			(* Case 60 - AspirazioneDX *)
			60: 
				IF AspirazioneSX^.Status.CommandDone AND AspirazioneDX^.Status.CommandDone THEN
					AspirazioneDX^.Command^.Aspirazione_ON 	:= FALSE;
					AspirazioneDX^.Command^.Aspirazione_OFF	:= FALSE;
					AspirazioneSX^.Command^.Aspirazione_ON 	:= FALSE;
					AspirazioneSX^.Command^.Aspirazione_OFF	:= FALSE;
					TFCommandCase(ADR(CmdExe),100,CommandCase_JMP);
				ELSIF AspirazioneSX^.Status.ErrorID <> ErrNULL THEN
					TFClearAllCmdModulePinzaCompleta(AspirazioneDX,AspirazioneSX,CilindroApertura,CilindroSbloccoRotazione,AspirazioneFaldaDX,AspirazioneFaldaSX);
					TFError(ErrCYLINDER,AspirazioneSX^.Status.ErrorID,ADR(CmdExe),ADR(State),ADR(Error),ADR(ErrorLog));
				ELSIF AspirazioneDX^.Status.ErrorID <> ErrNULL THEN
					TFClearAllCmdModulePinzaCompleta(AspirazioneDX,AspirazioneSX,CilindroApertura,CilindroSbloccoRotazione,AspirazioneFaldaDX,AspirazioneFaldaSX);
					TFError(ErrCYLINDER,AspirazioneDX^.Status.ErrorID,ADR(CmdExe),ADR(State),ADR(Error),ADR(ErrorLog));
				END_IF

			(* Case 70 - CilindroTasteggio *)
			70: 
				//IF CilindroTasteggio^.Status.CommandDone THEN
				//	CilindroTasteggio^.Command.Activation 		:= FALSE;
				//	CilindroTasteggio^.Command.Deactivation 	:= FALSE;
					TFCommandCase(ADR(CmdExe),100,CommandCase_JMP);
				//END_IF								
				
			(* Case 100 - End *)
			100:(* Clear All Output Here *)
				TFStateUpdate(ADR(State),StateMAN_END);
				TFCommandExeClear(ADR(CmdExe));

			ELSE
				TFError(ErrNOCMDCASE,ErrNULL,ADR(CmdExe),ADR(State),ADR(Error),ADR(ErrorLog));
		END_CASE;

		IF TFTimerDone(ADR(Timeout)) THEN
			TFClearAllCmdModulePinzaCompleta(AspirazioneDX,AspirazioneSX,CilindroApertura,CilindroSbloccoRotazione,AspirazioneFaldaDX,AspirazioneFaldaSX);
			TFError(ErrCMDTIMEOUT,ErrNULL,ADR(CmdExe),ADR(State),ADR(Error),ADR(ErrorLog));
		END_IF
	

	(* ******************************************************************************************************** *)
	(* PRELOAD - Presa del pezzo *)
	(* ******************************************************************************************************** *)
	CmdPRELOAD:
		CASE CmdExe.CmdCase OF
			
			(* Case 0 - Init Command*)
			0: 	TFStateUpdate(ADR(State),StatePRELOAD_RUN);
				TFTimerSet(ADR(Timeout),30000+200,TRUE);
				TFTimerSet(ADR(Timer),30000,TRUE);
				PrelievoSuCavallina := FALSE;
				StatoPinza.ElementoPrelevato := FALSE;
				IF TFCommandParRead(CmdExe.Cmd.Parameter,ADR(ParametersArray),2) THEN
					PrelievoSuCavallina	:= STRING_TO_BOOL(ParametersArray.Parameters[0]);
					AspiraSoloFalde		:= STRING_TO_BOOL(ParametersArray.Parameters[1]);
					TFCommandCase(ADR(CmdExe),10,CommandCase_JMP);
				ELSE
					TFError(ErrCMDPARNUM,ErrNULL,ADR(CmdExe),ADR(State),ADR(Error),ADR(ErrorLog));
					RETURN;
				END_IF;
				
			(* Case 10 - CilindroApertura *)
			10: 
				IF (ElementoInPrelievo.Typology = QUADROTTA OR ElementoInPrelievo.XDim >= 2700) AND AbilitaAperturaAutomaticaPinza THEN //sE HO LE CONDIZIONI APRO LA PINZA
					CilindroApertura^.Command.Activation 	:= TRUE;
					CilindroApertura^.Command.Deactivation 	:= FALSE;
	
					IF CilindroApertura^.Status.Active THEN
						CilindroApertura^.Command.Activation 	:= FALSE;
						CilindroApertura^.Command.Deactivation 	:= FALSE;
						TFCommandCase(ADR(CmdExe),20,CommandCase_JMP);
					ELSIF CilindroApertura^.Status.ErrorID <> ErrNULL THEN
						TFClearAllCmdModulePinzaCompleta(AspirazioneDX,AspirazioneSX,CilindroApertura,CilindroSbloccoRotazione,AspirazioneFaldaDX,AspirazioneFaldaSX);
						TFError(ErrCYLINDER,CilindroApertura^.Status.ErrorID,ADR(CmdExe),ADR(State),ADR(Error),ADR(ErrorLog));
					END_IF
				ELSE

					CilindroApertura^.Command.Activation 	:= FALSE;
					CilindroApertura^.Command.Deactivation 	:= TRUE;
	
					IF CilindroApertura^.Status.Inactive THEN
						CilindroApertura^.Command.Activation 	:= FALSE;
						CilindroApertura^.Command.Deactivation 	:= FALSE;
						TFCommandCase(ADR(CmdExe),20,CommandCase_JMP);
					ELSIF CilindroApertura^.Status.ErrorID <> ErrNULL THEN
						TFClearAllCmdModulePinzaCompleta(AspirazioneDX,AspirazioneSX,CilindroApertura,CilindroSbloccoRotazione,AspirazioneFaldaDX,AspirazioneFaldaSX);
						TFError(ErrCYLINDER,CilindroApertura^.Status.ErrorID,ADR(CmdExe),ADR(State),ADR(Error),ADR(ErrorLog));
					END_IF
					
				END_IF

			(* Case 20 - CilindroSbloccoRotazione *)
			20: 
				IF PrelievoSuCavallina THEN
					CilindroSbloccoRotazione^.Command.Activation 	:= AbilitazioneSbloccoRotazione;
					CilindroSbloccoRotazione^.Command.Deactivation 	:= FALSE;
	
					//CilindroTasteggio^.Command.Activation 		:= AbilitazioneCilindriTastatori;
					//CilindroTasteggio^.Command.Deactivation 	:= FALSE;
					
					IF (CilindroSbloccoRotazione^.Status.Active OR NOT AbilitazioneSbloccoRotazione) THEN
						CilindroSbloccoRotazione^.Command.Activation 	:= FALSE;
						CilindroSbloccoRotazione^.Command.Deactivation 	:= FALSE;
						//CilindroTasteggio^.Command.Activation 		:= FALSE;
						//CilindroTasteggio^.Command.Deactivation 	:= FALSE;
						TFCommandCase(ADR(CmdExe),30,CommandCase_JMP);
					ELSIF CilindroSbloccoRotazione^.Status.ErrorID <> ErrNULL AND AbilitazioneSbloccoRotazione THEN
						TFClearAllCmdModulePinzaCompleta(AspirazioneDX,AspirazioneSX,CilindroApertura,CilindroSbloccoRotazione,AspirazioneFaldaDX,AspirazioneFaldaSX);
						TFError(ErrCYLINDER,CilindroSbloccoRotazione^.Status.ErrorID,ADR(CmdExe),ADR(State),ADR(Error),ADR(ErrorLog));
					//ELSIF CilindroTasteggio^.Status.ErrorID <> ErrNULL THEN
					//	TFClearAllCmdModulePinzaCompleta(AspirazioneDX,AspirazioneSX,CilindroApertura,CilindroSbloccoRotazione,AspirazioneFaldaDX,AspirazioneFaldaSX);
					//	TFError(ErrCYLINDER,CilindroTasteggio^.Status.ErrorID,ADR(CmdExe),ADR(State),ADR(Error),ADR(ErrorLog));
					END_IF

				ELSE
					TFCommandCase(ADR(CmdExe),30,CommandCase_JMP);
				END_IF

			(* Case 30 - AspirazioneFaldaDX *)
			30: 

				IF NOT PrelievoSuCavallina AND AspiraSoloFalde THEN
					AspirazioneFaldaDX^.Command.Activation 	:= TRUE;
					AspirazioneFaldaDX^.Command.Deactivation 	:= FALSE;
					AspirazioneFaldaSX^.Command.Activation 	:= TRUE;
					AspirazioneFaldaSX^.Command.Deactivation 	:= FALSE;
					
					IF AspirazioneFaldaDX^.Status.Active AND AspirazioneFaldaSX^.Status.Active THEN
						AspirazioneFaldaDX^.Command.Activation 	:= FALSE;
						AspirazioneFaldaDX^.Command.Deactivation 	:= FALSE;
						AspirazioneFaldaSX^.Command.Activation 	:= FALSE;
						AspirazioneFaldaSX^.Command.Deactivation 	:= FALSE;
						TFCommandCase(ADR(CmdExe),40,CommandCase_JMP);
					ELSIF AspirazioneFaldaDX^.Status.ErrorID <> ErrNULL THEN
						TFClearAllCmdModulePinzaCompleta(AspirazioneDX,AspirazioneSX,CilindroApertura,CilindroSbloccoRotazione,AspirazioneFaldaDX,AspirazioneFaldaSX);
						TFError(ErrCYLINDER,AspirazioneFaldaDX^.Status.ErrorID,ADR(CmdExe),ADR(State),ADR(Error),ADR(ErrorLog));
					ELSIF AspirazioneFaldaSX^.Status.ErrorID <> ErrNULL THEN
						TFClearAllCmdModulePinzaCompleta(AspirazioneDX,AspirazioneSX,CilindroApertura,CilindroSbloccoRotazione,AspirazioneFaldaDX,AspirazioneFaldaSX);
						TFError(ErrCYLINDER,AspirazioneFaldaSX^.Status.ErrorID,ADR(CmdExe),ADR(State),ADR(Error),ADR(ErrorLog));
					END_IF
				ELSE
					TFCommandCase(ADR(CmdExe),40,CommandCase_JMP);
				END_IF


			(* Case 40 - AspirazioneDX + AspirazioneSX *)
			40: 
				AspirazioneDX^.Command^.Aspirazione_ON 	:= TRUE;
				AspirazioneDX^.Command^.Aspirazione_OFF := FALSE;
			
				AspirazioneSX^.Command^.Aspirazione_ON 	:= TRUE;
				AspirazioneSX^.Command^.Aspirazione_OFF := FALSE;
	
				IF AspirazioneDX^.Status.CommandDone AND AspirazioneSX^.Status.CommandDone THEN
					AspirazioneDX^.Command^.Aspirazione_ON 	:= FALSE;
					AspirazioneDX^.Command^.Aspirazione_OFF	:= FALSE;
					AspirazioneSX^.Command^.Aspirazione_ON 	:= FALSE;
					AspirazioneSX^.Command^.Aspirazione_OFF	:= FALSE;
					TFCommandCase(ADR(CmdExe),100,CommandCase_JMP);
				ELSIF AspirazioneSX^.Status.ErrorID <> ErrNULL THEN
					TFClearAllCmdModulePinzaCompleta(AspirazioneDX,AspirazioneSX,CilindroApertura,CilindroSbloccoRotazione,AspirazioneFaldaDX,AspirazioneFaldaSX);
					TFError(ErrCYLINDER,AspirazioneSX^.Status.ErrorID,ADR(CmdExe),ADR(State),ADR(Error),ADR(ErrorLog));
				ELSIF AspirazioneDX^.Status.ErrorID <> ErrNULL THEN
					TFClearAllCmdModulePinzaCompleta(AspirazioneDX,AspirazioneSX,CilindroApertura,CilindroSbloccoRotazione,AspirazioneFaldaDX,AspirazioneFaldaSX);
					TFError(ErrCYLINDER,AspirazioneDX^.Status.ErrorID,ADR(CmdExe),ADR(State),ADR(Error),ADR(ErrorLog));
				END_IF
				
			(* Case 100 *)
			100:TFStateUpdate(ADR(State),StatePRELOAD_END);
				TFCommandExeClear(ADR(CmdExe));

			ELSE
				TFError(ErrNOCMDCASE,ErrNULL,ADR(CmdExe),ADR(State),ADR(Error),ADR(ErrorLog));
		END_CASE

		IF TFTimerDone(ADR(Timeout)) THEN
			TFClearAllCmdModulePinzaCompleta(AspirazioneDX,AspirazioneSX,CilindroApertura,CilindroSbloccoRotazione,AspirazioneFaldaDX,AspirazioneFaldaSX);
			TFError(ErrCMDTIMEOUT,ErrNULL,ADR(CmdExe),ADR(State),ADR(Error),ADR(ErrorLog));
		END_IF
	


	(* ******************************************************************************************************** *)
	(* LOAD - Presa del pezzo *)
	(* ******************************************************************************************************** *)
	CmdCHECKPRESENCE:
		CASE CmdExe.CmdCase OF
			
			(* Case 0 - Init Command*)
			0: 	TFStateUpdate(ADR(State),StateCHECKPRESENCE_RUN);
				TFTimerSet(ADR(Timeout),60000.0+100+HMI_TempoControlloPresaPiastrella,TRUE);
				TFTimerSet(ADR(Timer),2000.0+HMI_TempoControlloPresaPiastrella,TRUE);
				TFTimerSet(ADR(TimerPresaPiastrella),HMI_TempoControlloPresaPiastrella,TRUE);
				StatoPinza.ElementoPrelevato := FALSE;
				CilindroSbloccoRotazione^.Command.Activation 	:= FALSE;
				CilindroSbloccoRotazione^.Command.Deactivation 	:= TRUE;

				TFCommandCase(ADR(CmdExe),1,CommandCase_INC);
				
			(* Case 1 - *)					
			1:
				StatoPinza.ElementoPrelevato := FALSE;
				IF CilindroSbloccoRotazione^.Status.Inactive THEN //Attendo un tempo impostatato da HMI per attendere che la piastrella sia veramente in presa
					CilindroSbloccoRotazione^.Command.Activation 	:= FALSE;
					CilindroSbloccoRotazione^.Command.Deactivation 	:= TRUE;	
				END_IF

			IF IN.ByPassSensoreVuoto OR TFTimerDone(ADR(TimerPresaPiastrella)) THEN 
					//Tutte piastrelle o tutte falde
					IF (AspirazioneDX^.Status.DepressioneSoglia1_OK AND AspirazioneSX^.Status.DepressioneSoglia1_OK) OR
						((AspirazioneFaldaDX^.Status.Active AND IN.TastoreCartoneDX AND FTC_FaldaDXFiltrata) AND
						(AspirazioneFaldaSX^.Status.Active AND IN.TastoreCartoneSX AND FTC_FaldaSXFiltrata)) OR
						IN.ByPassSensoreVuoto THEN
							StatoPinza.ElementoPrelevato := TRUE;
							TFCommandCase(ADR(CmdExe),1,CommandCase_INC);
					ELSIF TFTimerDone(ADR(TimerPresaPiastrella)) THEN
						TFCommandCase(ADR(CmdExe),1,CommandCase_INC);
						StatoPinza.ElementoPrelevato := FALSE;	
					END_IF			
				ELSIF TFTimerDone(ADR(TimerPresaPiastrella)) THEN
					TFCommandCase(ADR(CmdExe),1,CommandCase_INC);
					StatoPinza.ElementoPrelevato := FALSE;
				END_IF			
				IF TFTimerDone(ADR(Timer)) THEN
					TFClearAllCmdModulePinzaCompleta(AspirazioneDX,AspirazioneSX,CilindroApertura,CilindroSbloccoRotazione,AspirazioneFaldaDX,AspirazioneFaldaSX);
					TFError(ErrMalfunzionamentoSensoriPresenzaPinza,ErrNULL,ADR(CmdExe),ADR(State),ADR(Error),ADR(ErrorLog));
				ELSIF TFTimerDone(ADR(Timeout)) THEN
					TFClearAllCmdModulePinzaCompleta(AspirazioneDX,AspirazioneSX,CilindroApertura,CilindroSbloccoRotazione,AspirazioneFaldaDX,AspirazioneFaldaSX);
					TFError(ErrCMDTIMEOUT,ErrNULL,ADR(CmdExe),ADR(State),ADR(Error),ADR(ErrorLog));
				END_IF
		
			(* Case 2 - *)		
			2: 
				TFTimerSet(ADR(TimerAspirazione),1,TRUE);
				TFCommandCase(ADR(CmdExe),1,CommandCase_INC);
				IF TFTimerDone(ADR(Timer)) THEN
					TFClearAllCmdModulePinzaCompleta(AspirazioneDX,AspirazioneSX,CilindroApertura,CilindroSbloccoRotazione,AspirazioneFaldaDX,AspirazioneFaldaSX);
					TFError(ErrMalfunzionamentoSensoriPresenzaPinza,ErrNULL,ADR(CmdExe),ADR(State),ADR(Error),ADR(ErrorLog));
				ELSIF TFTimerDone(ADR(Timeout)) THEN
					TFClearAllCmdModulePinzaCompleta(AspirazioneDX,AspirazioneSX,CilindroApertura,CilindroSbloccoRotazione,AspirazioneFaldaDX,AspirazioneFaldaSX);
					TFError(ErrCMDTIMEOUT,ErrNULL,ADR(CmdExe),ADR(State),ADR(Error),ADR(ErrorLog));
				END_IF				
				
			3:
				IF TFTimerDone(ADR(TimerAspirazione)) THEN
					TFStateUpdate(ADR(State),StateCHECKPRESENCE_RUN+10);
					TFCommandCase(ADR(CmdExe),100,CommandCase_JMP);
				END_IF
				
			4:			
				IF 	((AspirazioneFaldaDX^.Status.Active AND IN.TastoreCartoneDX AND FTC_FaldaDXFiltrata AND NOT AspirazioneDX^.Status.DepressioneSoglia1_OK) OR
					(AspirazioneFaldaSX^.Status.Active AND IN.TastoreCartoneSX AND FTC_FaldaSXFiltrata AND NOT AspirazioneSX^.Status.DepressioneSoglia1_OK)) THEN
					StatoPinza.ElementoPrelevato := TRUE;
					TFCommandCase(ADR(CmdExe),100,CommandCase_JMP);
				ELSE
					TFCommandCase(ADR(CmdExe),100,CommandCase_JMP);
					StatoPinza.ElementoPrelevato := FALSE;
				END_IF	
			
			10:	
				IF NOT	StatoPinza.ElementoPrelevato THEN
					IF (AspirazioneDX^.Status.DepressioneSoglia1_OK AND (IN.TastoreCartoneSX AND (FTC_FaldaSXFiltrata OR AspirazioneFaldaSX^.Status.Inactive)) AND NOT AspirazioneSX^.Status.DepressioneSoglia1_OK) THEN
						
						AspirazioneDX^.Command^.Aspirazione_ON 	:= FALSE;
						AspirazioneDX^.Command^.Aspirazione_OFF := FALSE;
						AspirazioneFaldaSX^.Command.Activation 		:= FALSE;
						AspirazioneFaldaSX^.Command.Deactivation 	:= TRUE;
						IF AspirazioneFaldaSX^.Status.Inactive THEN
							AspirazioneFaldaSX^.Command.Activation 		:= FALSE;
							AspirazioneFaldaSX^.Command.Deactivation 	:= FALSE;
							AspirazioneFaldaSX^.Command.Activation 		:= FALSE;
							AspirazioneFaldaSX^.Command.Deactivation 	:= FALSE;

							//TFTimerSet(ADR(TimerAspirazione),HMI_TempoRilascioInDeposito,TRUE);
							TFCommandCase(ADR(CmdExe),12,CommandCase_JMP);
						ELSIF AspirazioneSX^.Status.ErrorID <> ErrNULL THEN
							TFClearAllCmdModulePinzaCompleta(AspirazioneDX,AspirazioneSX,CilindroApertura,CilindroSbloccoRotazione,AspirazioneFaldaDX,AspirazioneFaldaSX);
							TFError(ErrCYLINDER,AspirazioneSX^.Status.ErrorID,ADR(CmdExe),ADR(State),ADR(Error),ADR(ErrorLog));
						ELSIF AspirazioneDX^.Status.ErrorID <> ErrNULL THEN
							TFClearAllCmdModulePinzaCompleta(AspirazioneDX,AspirazioneSX,CilindroApertura,CilindroSbloccoRotazione,AspirazioneFaldaDX,AspirazioneFaldaSX);
							TFError(ErrCYLINDER,AspirazioneDX^.Status.ErrorID,ADR(CmdExe),ADR(State),ADR(Error),ADR(ErrorLog));
						END_IF
		
					ELSIF (AspirazioneSX^.Status.DepressioneSoglia1_OK AND (IN.TastoreCartoneDX AND (FTC_FaldaDXFiltrata OR AspirazioneFaldaDX^.Status.Inactive)) AND NOT AspirazioneDX^.Status.DepressioneSoglia1_OK) THEN
											
						AspirazioneFaldaDX^.Command.Activation 		:= FALSE;
						AspirazioneFaldaDX^.Command.Deactivation 	:= TRUE;
						IF AspirazioneFaldaDX^.Status.Inactive THEN
							AspirazioneFaldaDX^.Command.Activation 		:= FALSE;
							AspirazioneFaldaDX^.Command.Deactivation 	:= FALSE;
							AspirazioneFaldaSX^.Command.Activation 		:= FALSE;
							AspirazioneFaldaSX^.Command.Deactivation 	:= FALSE;

							//TFTimerSet(ADR(TimerAspirazione),HMI_TempoRilascioInDeposito,TRUE);
							TFCommandCase(ADR(CmdExe),12,CommandCase_JMP);
						ELSIF AspirazioneSX^.Status.ErrorID <> ErrNULL THEN
							TFClearAllCmdModulePinzaCompleta(AspirazioneDX,AspirazioneSX,CilindroApertura,CilindroSbloccoRotazione,AspirazioneFaldaDX,AspirazioneFaldaSX);
							TFError(ErrCYLINDER,AspirazioneSX^.Status.ErrorID,ADR(CmdExe),ADR(State),ADR(Error),ADR(ErrorLog));
						ELSIF AspirazioneDX^.Status.ErrorID <> ErrNULL THEN
							TFClearAllCmdModulePinzaCompleta(AspirazioneDX,AspirazioneSX,CilindroApertura,CilindroSbloccoRotazione,AspirazioneFaldaDX,AspirazioneFaldaSX);
							TFError(ErrCYLINDER,AspirazioneDX^.Status.ErrorID,ADR(CmdExe),ADR(State),ADR(Error),ADR(ErrorLog));
						END_IF
						
					ELSIF (((AspirazioneFaldaDX^.Status.Active AND IN.TastoreCartoneDX AND NOT FTC_FaldaDXFiltrata AND NOT AspirazioneDX^.Status.DepressioneSoglia1_OK)) AND
						(AspirazioneFaldaSX^.Status.Active AND IN.TastoreCartoneSX AND NOT FTC_FaldaSXFiltrata AND NOT AspirazioneSX^.Status.DepressioneSoglia1_OK)) THEN
							TFCommandCase(ADR(CmdExe),1,CommandCase_INC);	

					END_IF
					//TFCommandCase(ADR(CmdExe),4,CommandCase_JMP);
				
				ELSE
					TFCommandCase(ADR(CmdExe),1,CommandCase_INC);
				END_IF
				IF TFTimerDone(ADR(Timer)) THEN
					TFClearAllCmdModulePinzaCompleta(AspirazioneDX,AspirazioneSX,CilindroApertura,CilindroSbloccoRotazione,AspirazioneFaldaDX,AspirazioneFaldaSX);
					TFError(ErrMalfunzionamentoSensoriPresenzaPinza,ErrNULL,ADR(CmdExe),ADR(State),ADR(Error),ADR(ErrorLog));
				ELSIF TFTimerDone(ADR(Timeout)) THEN
					TFClearAllCmdModulePinzaCompleta(AspirazioneDX,AspirazioneSX,CilindroApertura,CilindroSbloccoRotazione,AspirazioneFaldaDX,AspirazioneFaldaSX);
					TFError(ErrCMDTIMEOUT,ErrNULL,ADR(CmdExe),ADR(State),ADR(Error),ADR(ErrorLog));
				END_IF
				
			11:
				IF TFTimerDone(ADR(TimerAspirazione)) THEN
					TFStateUpdate(ADR(State),StateCHECKPRESENCE_RUN+10);
					TFCommandCase(ADR(CmdExe),100,CommandCase_JMP);
				END_IF
				
			12:			
				IF 	(IN.TastoreCartoneDX AND NOT FTC_FaldaDXFiltrata AND AspirazioneSX^.Status.DepressioneSoglia1_OK) OR
					(IN.TastoreCartoneSX AND NOT FTC_FaldaSXFiltrata AND AspirazioneDX^.Status.DepressioneSoglia1_OK) THEN
					StatoPinza.ElementoPrelevato := TRUE;
					TFCommandCase(ADR(CmdExe),100,CommandCase_JMP);
				ELSE
					TFCommandCase(ADR(CmdExe),100,CommandCase_JMP);
					StatoPinza.ElementoPrelevato := FALSE;
				END_IF	
				
				
			(* Case 100 *)
			100:TFStateUpdate(ADR(State),StateCHECKPRESENCE_END);
				TFCommandExeClear(ADR(CmdExe));

			ELSE
				TFError(ErrNOCMDCASE,ErrNULL,ADR(CmdExe),ADR(State),ADR(Error),ADR(ErrorLog));
		END_CASE
				
	
	(* ******************************************************************************************************** *)
	(* UNLOAD - Attivazione aspirazione + discesa ventose *)
	(* ******************************************************************************************************** *)
	CmdUNLOAD:
		CASE CmdExe.CmdCase OF
			
			(* Case 0 - Init Command*)
			0: 	TFStateUpdate(ADR(State),StateUNLOAD_RUN);
				TFTimerSet(ADR(Timeout),30000+200,TRUE);
				TFTimerSet(ADR(Timer),30000,TRUE);
				DisattivazioneTotaleAspirazioni := FALSE;
				
				IF Mission^.State = MISSION_STATE_DEPOSITO_FALDA_DEPAL_RUN THEN
					TFCommandCase(ADR(CmdExe),10,CommandCase_JMP);
				ELSIF Mission^.State = MISSION_STATE_DEPOSITO_LASTRA_DEPAL_RUN THEN
		
					IF NOT StatoPinza.LatoDxFaldaInPresa AND NOT StatoPinza.LatoSxFaldaInPresa THEN
						StatoPinza.ElementoPrelevato := FALSE;
						DisattivazioneTotaleAspirazioni := TRUE;
						TFCommandCase(ADR(CmdExe),10,CommandCase_JMP);
					ELSE
						TFCommandCase(ADR(CmdExe),20,CommandCase_JMP);
					END_IF					
				ELSE
					DisattivazioneTotaleAspirazioni := TRUE;
					StatoPinza.ElementoPrelevato := FALSE;
					TFCommandCase(ADR(CmdExe),10,CommandCase_JMP);
				END_IF
				
			(* Case 10 - Disattivazione Aspirazione falde *)					
			10:	
				AspirazioneFaldaDX^.Command.Activation 		:= FALSE;
				AspirazioneFaldaDX^.Command.Deactivation 	:= TRUE;
				AspirazioneFaldaSX^.Command.Activation 		:= FALSE;
				AspirazioneFaldaSX^.Command.Deactivation 	:= TRUE;

				CilindroSbloccoRotazione^.Command.Activation 	:= FALSE;
				CilindroSbloccoRotazione^.Command.Deactivation 	:= TRUE;
				
				IF AspirazioneFaldaDX^.Status.Inactive AND AspirazioneFaldaSX^.Status.Inactive AND CilindroSbloccoRotazione^.Status.Inactive THEN
					AspirazioneFaldaDX^.Command.Activation 		:= FALSE;
					AspirazioneFaldaDX^.Command.Deactivation 	:= FALSE;
					AspirazioneFaldaSX^.Command.Activation 		:= FALSE;
					AspirazioneFaldaSX^.Command.Deactivation 	:= FALSE;
					CilindroSbloccoRotazione^.Command.Activation 	:= FALSE;
					CilindroSbloccoRotazione^.Command.Deactivation 	:= FALSE;
					IF DisattivazioneTotaleAspirazioni THEN
						TFCommandCase(ADR(CmdExe),20,CommandCase_JMP);
					ELSE
						TFCommandCase(ADR(CmdExe),100,CommandCase_JMP);
					END_IF				
				ELSIF AspirazioneFaldaDX^.Status.ErrorID <> ErrNULL THEN
					TFClearAllCmdModulePinzaCompleta(AspirazioneDX,AspirazioneSX,CilindroApertura,CilindroSbloccoRotazione,AspirazioneFaldaDX,AspirazioneFaldaSX);
					TFError(ErrCYLINDER,AspirazioneFaldaDX^.Status.ErrorID,ADR(CmdExe),ADR(State),ADR(Error),ADR(ErrorLog));
				ELSIF AspirazioneFaldaSX^.Status.ErrorID <> ErrNULL THEN
					TFClearAllCmdModulePinzaCompleta(AspirazioneDX,AspirazioneSX,CilindroApertura,CilindroSbloccoRotazione,AspirazioneFaldaDX,AspirazioneFaldaSX);
					TFError(ErrCYLINDER,AspirazioneFaldaSX^.Status.ErrorID,ADR(CmdExe),ADR(State),ADR(Error),ADR(ErrorLog));
				ELSIF CilindroSbloccoRotazione^.Status.ErrorID <> ErrNULL THEN
					TFClearAllCmdModulePinzaCompleta(AspirazioneDX,AspirazioneSX,CilindroApertura,CilindroSbloccoRotazione,AspirazioneFaldaDX,AspirazioneFaldaSX);
					TFError(ErrCYLINDER,CilindroSbloccoRotazione^.Status.ErrorID,ADR(CmdExe),ADR(State),ADR(Error),ADR(ErrorLog));
				END_IF
			
			(* Case 20 - Disattivazione aspirazione piastrella *)		
			20: 
				AspirazioneDX^.Command^.Aspirazione_ON 	:= FALSE;
				AspirazioneDX^.Command^.Aspirazione_OFF := TRUE;
			
				AspirazioneSX^.Command^.Aspirazione_ON 	:= FALSE;
				AspirazioneSX^.Command^.Aspirazione_OFF := TRUE;
		
				IF AspirazioneDX^.Status.CommandDone AND AspirazioneSX^.Status.CommandDone THEN
					AspirazioneDX^.Command^.Aspirazione_ON 	:= FALSE;
					AspirazioneDX^.Command^.Aspirazione_OFF	:= FALSE;
					AspirazioneSX^.Command^.Aspirazione_ON 	:= FALSE;
					AspirazioneSX^.Command^.Aspirazione_OFF	:= FALSE;
					TFTimerSet(ADR(TimerAspirazione),HMI_TempoRilascioInDeposito,TRUE);
					TFCommandCase(ADR(CmdExe),30,CommandCase_JMP);
				ELSIF AspirazioneSX^.Status.ErrorID <> ErrNULL THEN
					TFClearAllCmdModulePinzaCompleta(AspirazioneDX,AspirazioneSX,CilindroApertura,CilindroSbloccoRotazione,AspirazioneFaldaDX,AspirazioneFaldaSX);
					TFError(ErrCYLINDER,AspirazioneSX^.Status.ErrorID,ADR(CmdExe),ADR(State),ADR(Error),ADR(ErrorLog));
				ELSIF AspirazioneDX^.Status.ErrorID <> ErrNULL THEN
					TFClearAllCmdModulePinzaCompleta(AspirazioneDX,AspirazioneSX,CilindroApertura,CilindroSbloccoRotazione,AspirazioneFaldaDX,AspirazioneFaldaSX);
					TFError(ErrCYLINDER,AspirazioneDX^.Status.ErrorID,ADR(CmdExe),ADR(State),ADR(Error),ADR(ErrorLog));
				END_IF
			
			(* Case 30 - Attesa tempo distacco *)		
			30:
				IF TFTimerDone(ADR(TimerAspirazione)) THEN
					IF IN.RichiestaRicalibrazioneOvemEsterna AND NOT IN.ByPassSensoreVuoto THEN
						IN.RichiestaRicalibrazioneOvemEsterna := FALSE;
						TFCommandCase(ADR(CmdExe),40,CommandCase_JMP);
					ELSE
						TFCommandCase(ADR(CmdExe),100,CommandCase_JMP);
					END_IF		
				END_IF
				
			(* Case 40 - Attesa tempo distacco *)		
			40:	
				AspirazioneDX^.Command^.Aspirazione_ON_ScritturaSoglia 	:= TRUE;
				AspirazioneSX^.Command^.Aspirazione_ON_ScritturaSoglia 	:= TRUE;
				IF AspirazioneDX^.Status.CommandDone AND AspirazioneSX^.Status.CommandDone THEN
					AspirazioneDX^.Command^.Aspirazione_ON_ScritturaSoglia		:= FALSE;
					AspirazioneSX^.Command^.Aspirazione_ON_ScritturaSoglia		:= FALSE;
					TFCommandCase(ADR(CmdExe),100,CommandCase_JMP);
				ELSIF TFTimerDone(ADR(Timer)) THEN
					AspirazioneDX^.Command^.Aspirazione_ON_ScritturaSoglia		:= FALSE;
					AspirazioneSX^.Command^.Aspirazione_ON_ScritturaSoglia		:= FALSE;
					TFError(ErrTOHOME,ErrNULL,ADR(CmdExe),ADR(State),ADR(Error),ADR(ErrorLog));
				END_IF
				
		
			(* Case 100 *)
			100:TFStateUpdate(ADR(State),StateUNLOAD_END);
				TFCommandExeClear(ADR(CmdExe));

			ELSE
				TFError(ErrNOCMDCASE,ErrNULL,ADR(CmdExe),ADR(State),ADR(Error),ADR(ErrorLog));
		END_CASE

		IF TFTimerDone(ADR(Timeout)) THEN
			TFClearAllCmdModulePinzaCompleta(AspirazioneDX,AspirazioneSX,CilindroApertura,CilindroSbloccoRotazione,AspirazioneFaldaDX,AspirazioneFaldaSX);
			TFError(ErrCMDTIMEOUT,ErrNULL,ADR(CmdExe),ADR(State),ADR(Error),ADR(ErrorLog));
		END_IF


	ELSE
		TFError(ErrNOCMD,ErrNULL,ADR(CmdExe),ADR(State),ADR(Error),ADR(ErrorLog));

END_CASE;


(* ******************************************************************************************************** *)
(* State Input/Output *)
(* ******************************************************************************************************** *)
(* Fill Input/Output bit with sensor, electrovalve, etc. status *)

StatoPinza.LatoDxAperto 			:= CilindroApertura^.Status.Active;
StatoPinza.LatoDxChiuso 			:= CilindroApertura^.Status.Inactive;
StatoPinza.LatoSxAperto				:= CilindroApertura^.Status.Active;
StatoPinza.LatoSxChiuso				:= CilindroApertura^.Status.Inactive;

StatoPinza.LatoDxFaldaInPresa		:= AspirazioneFaldaDX^.Status.Active AND IN.TastoreCartoneDX AND NOT AspirazioneDX^.Status.DepressioneSoglia1_OK AND FTC_FaldaDXFiltrata;
StatoPinza.LatoDxPiastrellaInPresa	:= (AspirazioneDX^.Status.DepressioneSoglia1_OK  OR (IN.ByPassSensoreVuoto AND StatoPinza.ElementoPrelevato));// AND NOT IN.TastoreCartoneDX;
StatoPinza.LatoSxFaldaInPresa		:= AspirazioneFaldaSX^.Status.Active AND IN.TastoreCartoneSX AND NOT AspirazioneSX^.Status.DepressioneSoglia1_OK AND FTC_FaldaSXFiltrata;
StatoPinza.LatoSxPiastrellaInPresa	:=(AspirazioneSX^.Status.DepressioneSoglia1_OK  OR (IN.ByPassSensoreVuoto AND StatoPinza.ElementoPrelevato));// AND  IN.TastoreCartoneSX;
StatoPinza.RotazioneBloccata		:= CilindroSbloccoRotazione^.Status.Inactive;
StatoPinza.RotazioneSbloccata 		:= CilindroSbloccoRotazione^.Status.Active;

(* ******************************************************************************************************** *)
(* Input *)
(* ******************************************************************************************************** *)

(* ******************************************************************************************************** *)
(* Alarm *)
(* ******************************************************************************************************** *)

(* ******************************************************************************************************** *)
(* Error Check - Clear All Output!!! *)
(* ******************************************************************************************************** *)
IF Error.Code > ErrNULL THEN
	IF CmdExe.Code <> CmdNOP THEN
		IF CmdExe.Code <> CmdSTOP AND
			CmdExe.Code <> CmdPOWER AND
			CmdExe.Code <> CmdRESET AND
			CmdExe.Code <> CmdMAN AND
			CmdExe.Code <> CmdLOAD AND
			CmdExe.Code <> CmdUNLOAD THEN
			TFCommandClear(ADR(CmdNext));
			TFCommandExeClear(ADR(CmdExe));

			(* Clear All Output Here *)

		END_IF;
	END_IF;
END_IF;


(* ******************************************************************************************************** *)
(* Common Outputs *)
(* ******************************************************************************************************** *)

END_FUNCTION_BLOCK

// ---- POUs/TFModules/Moduli TF/TFModulePalletizer_Pinza_Semplice.TcPOU
FUNCTION_BLOCK TFModulePalletizer_Pinza_Semplice
VAR_INPUT
	Cmd : CommandBuffer;
	Cfg : Config;
	IN : TFMchinePalletizer_PinzaVentose_IN;
		
	IN_Ax : Module_Palletizer_Ax_IN;
	
	AspirazioneDX : POINTER TO TF_VacumOVEM;
	AspirazioneSX : POINTER TO TF_VacumOVEM;

	ModuleJ : POINTER TO TFModulePalletizer_Ax;

	ManCmd 				: POINTER TO TFMachinePalletizer_PinzaVentoseManCmd;
	ElementoInPrelievo 	: TFMachinePalletizer_PlaceElement;
	DataElement			: TFMachinePalletizer_DataElement; (* Struttura dati che la macchina acquisisce/trasferisce in fase di pallettizzazione/depallettizazione *)
	PrelievoSuCavallina : BOOL;//indica che il prelievo è su cavallina
	AbilitazioneCilindriTastatori : bool;

	Mission : POINTER TO TFMachinePalletizer_Mission;
	AbilitazioneSbloccoRotazione 	: BOOL;//Abilitazione sblocco pinza
	AbilitaAperturaAutomaticaPinza : BOOL;//Abilitazione apertura automatica pinza
	PrelivoDaPalletSingoloConFalde : BOOL;
	AbilitaPrioritaPrelPiasterllaPianiSfalsati : bool;
END_VAR
VAR_OUTPUT
	CmdExe : CommandExe;
	CmdExd : CommandExe;
	CmdNext : Command;
	CmdLog : CommandLog;
	ProgramLog : ProgrammaLog; 
	State : State;
	StateLog : StateLog;
	Error : Error;
	ErrorLog : ErrorLog;
	Warning : Warning;
	WarningLog : WarningLog;
	OUT : TFMachinePalletizer_PinzaVentose_OUT;
	StatoPinza : TFMachinePalletizer_PinzaState;

END_VAR
VAR
	Power : UINT;
	Init : BOOL;
	Timer : REAL;
	Timeout : REAL;
	TimerAspirazione : REAL;
	ParametersArray : ParametersArray;
	MAN_Actuator : UINT;
	MAN_Cmd : UINT;

	DistanzaFTC0 : REAL;
	DistanzaFTC180 : REAL;

	TimerPresaPiastrella : REAL;		
	DisattivazioneTotaleAspirazioni : bool;
	FiltroFTCFaldaSX : Signal_Filter;
	FiltroFTCFaldaDX : Signal_Filter;
	
	FTC_FaldaSXFiltrata : BOOL;
	FTC_FaldaDXFiltrata : bool;
	
	PostazionePrelievo : int;
END_VAR

IF NOT Init THEN
	TFCommandBufferClear(ADR(Cmd));
	TFCommandClear(ADR(CmdNext));
	TFCommandExeClear(ADR(CmdExe));
	TFStateUpdate(ADR(State),StateNOP);
	TFErrorClear(ADR(Error));
	TFWarningClear(ADR(Warning));
	Init := TRUE;
	CmdExe.Code := 1;
END_IF

(* Generic Timer - Add here all your Timers *)
TFTimerCall(ADR(Timer),Cfg.TimeBase);
TFTimerCall(ADR(Timeout),Cfg.TimeBase);
TFTimerCall(ADR(TimerPresaPiastrella),Cfg.TimeBase);
TFTimerCall(ADR(TimerAspirazione),Cfg.TimeBase);
(* External To Buffered Command *)
TFCommandToNext(ADR(Cmd),ADR(CmdNext),ADR(CmdExe),ADR(Cfg),ADR(Error),ADR(ErrorLog),ADR(State));

(* Buffered To Exe Command *)
TFCommandToExecution(ADR(CmdNext),ADR(CmdExe),ADR(Error),ADR(ErrorLog),ADR(State),ADR(CmdLog));

(* Chiamata FB *)
AspirazioneDX^();
AspirazioneSX^();

CASE Mission^.PPick OF
	
	1: PostazionePrelievo := RullP1;
	
	2: PostazionePrelievo := RullP2;

END_CASE


(* Exe Command *)
CASE CmdExe.Code OF

	(* ******************************************************************************************************** *)
	(* Nop  *)
	(* ******************************************************************************************************** *)
	CmdNOP:	;			
	(* ******************************************************************************************************** *)
	(* Stop *)
	(* ******************************************************************************************************** *)
	CmdSTOP:
		CASE CmdExe.CmdCase OF
			
			(* Case 0 *)
			0: 	TFStateUpdate(ADR(State),StateSTOP_RUN);
				TFTimerSet(ADR(Timeout),500,TRUE);
				TFCommandCase(ADR(CmdExe),1,CommandCase_INC);

			(* Case 1 - Clear All Commands*)
			1:	
				TFCommandCase(ADR(CmdExe),100,CommandCase_JMP);
			(* Case 100 *)
			100:TFStateUpdate(ADR(State),StateSTOP_END);
				TFCommandExeClear(ADR(CmdExe));

			ELSE
				TFError(ErrNOCMDCASE,ErrNULL,ADR(CmdExe),ADR(State),ADR(Error),ADR(ErrorLog));
		END_CASE;
	
	(* ******************************************************************************************************** *)
	(* Error Reset *)
	(* ******************************************************************************************************** *)
	CmdRESET:
		CASE CmdExe.CmdCase OF

			(* Case 0 *)
			0: 	TFStateUpdate(ADR(State),StateRESET_RUN);
				TFTimerSet(ADR(Timeout),2000+100,TRUE);
				TFTimerSet(ADR(Timer),2000,TRUE);
				TFCommandCase(ADR(CmdExe),1,CommandCase_INC);
			
			(* Case 1 - RESET COMANDI*)
			1: 
				TFClearAllCmdModulePinza(AspirazioneDX,AspirazioneSX);
				TFCommandCase(ADR(CmdExe),1,CommandCase_INC);
			
			(* Case 2 - Invio comando di reset *)
			2:
				AspirazioneDX^.Command^.ErrorReset 				:= TRUE;	
				AspirazioneSX^.Command^.ErrorReset 				:= TRUE;	
				TFCommandCase(ADR(CmdExe),1,CommandCase_INC);
			
			(* Case 3 - Invio comando di reset *)
			3:
				IF AspirazioneDX^.Status.ErrorResetDone AND
					AspirazioneSX^.Status.ErrorResetDone THEN					
					TFClearAllCmdModulePinza(AspirazioneDX,AspirazioneSX);
					TFCommandCase(ADR(CmdExe),99,CommandCase_JMP);
				ELSIF TFTimerDone(ADR(Timer)) THEN
					TFClearAllCmdModulePinza(AspirazioneDX,AspirazioneSX);
					TFError(ErrTORESET,ErrNULL,ADR(CmdExe),ADR(State),ADR(Error),ADR(ErrorLog));
				END_IF

			(* Case 99 *)
			99:	TFErrorClear(ADR(Error));
				TFWarningClear(ADR(Warning));
				TFCommandCase(ADR(CmdExe),100,CommandCase_JMP);

			(* Case 100 *)
			100:TFStateUpdate(ADR(State),StateRESET_END);
				TFCommandExeClear(ADR(CmdExe));

			ELSE
				TFError(ErrNOCMDCASE,ErrNULL,ADR(CmdExe),ADR(State),ADR(Error),ADR(ErrorLog));
		END_CASE;

		(*IF AspirazioneDX^.Status.ErrorID <> ErrNULL THEN
			TFClearAllCmdModulePinza(AspirazioneDX,AspirazioneSX,CilindroApertura,CilindroSbloccoRotazione,AspirazioneFaldaDX,AspirazioneFaldaSX,CilindroTasteggio);
			TFError(ErrCYLINDER,AspirazioneDX^.Status.ErrorID,ADR(CmdExe),ADR(State),ADR(Error),ADR(ErrorLog));
		ELSIF AspirazioneSX^.Status.ErrorID <> ErrNULL THEN
			TFClearAllCmdModulePinza(AspirazioneDX,AspirazioneSX,CilindroApertura,CilindroSbloccoRotazione,AspirazioneFaldaDX,AspirazioneFaldaSX,CilindroTasteggio);
			TFError(ErrCYLINDER,AspirazioneSX^.Status.ErrorID,ADR(CmdExe),ADR(State),ADR(Error),ADR(ErrorLog));
		ELSIF CilindroApertura^.Status.ErrorID <> ErrNULL THEN
			TFClearAllCmdModulePinza(AspirazioneDX,AspirazioneSX,CilindroApertura,CilindroSbloccoRotazione,AspirazioneFaldaDX,AspirazioneFaldaSX,CilindroTasteggio);
			TFError(ErrCYLINDER,CilindroApertura^.Status.ErrorID,ADR(CmdExe),ADR(State),ADR(Error),ADR(ErrorLog));
		ELSIF CilindroSbloccoRotazione^.Status.ErrorID <> ErrNULL THEN
			TFClearAllCmdModulePinza(AspirazioneDX,AspirazioneSX,CilindroApertura,CilindroSbloccoRotazione,AspirazioneFaldaDX,AspirazioneFaldaSX,CilindroTasteggio);
			TFError(ErrCYLINDER,CilindroSbloccoRotazione^.Status.ErrorID,ADR(CmdExe),ADR(State),ADR(Error),ADR(ErrorLog));
		ELSIF AspirazioneFaldaDX^.Status.ErrorID <> ErrNULL THEN
			TFClearAllCmdModulePinza(AspirazioneDX,AspirazioneSX,CilindroApertura,CilindroSbloccoRotazione,AspirazioneFaldaDX,AspirazioneFaldaSX,CilindroTasteggio);
			TFError(ErrCYLINDER,AspirazioneFaldaDX^.Status.ErrorID,ADR(CmdExe),ADR(State),ADR(Error),ADR(ErrorLog));
		ELSIF AspirazioneFaldaSX^.Status.ErrorID <> ErrNULL THEN
			TFClearAllCmdModulePinza(AspirazioneDX,AspirazioneSX,CilindroApertura,CilindroSbloccoRotazione,AspirazioneFaldaDX,AspirazioneFaldaSX,CilindroTasteggio);
			TFError(ErrCYLINDER,AspirazioneFaldaSX^.Status.ErrorID,ADR(CmdExe),ADR(State),ADR(Error),ADR(ErrorLog));
		*)
		IF TFTimerDone(ADR(Timeout)) THEN
			TFClearAllCmdModulePinza(AspirazioneDX,AspirazioneSX);
			TFError(ErrCMDTIMEOUT,ErrNULL,ADR(CmdExe),ADR(State),ADR(Error),ADR(ErrorLog));
		END_IF
	
	(* ******************************************************************************************************** *)
	(* Power *)
	(* ******************************************************************************************************** *)
	CmdPOWER:
		CASE CmdExe.CmdCase OF
			
			(* Case 0 *)
			0: 	TFStateUpdate(ADR(State),StatePOWER_RUN);
				TFTimerSet(ADR(Timeout),500,TRUE);
				TFCommandCase(ADR(CmdExe),100,CommandCase_JMP);

			1: TFCommandCase(ADR(CmdExe),100,CommandCase_JMP);
			(* Case 100 *)
			100:TFStateUpdate(ADR(State),StatePOWER_END);
				TFCommandExeClear(ADR(CmdExe));

			ELSE
				TFError(ErrNOCMDCASE,ErrNULL,ADR(CmdExe),ADR(State),ADR(Error),ADR(ErrorLog));
		END_CASE
	
	(* ******************************************************************************************************** *)
	(* Home *)
	(* ******************************************************************************************************** *)
	CmdHOME:
		CASE CmdExe.CmdCase OF

			(* Case 0 *)
			0: 	TFStateUpdate(ADR(State),StateHOME_RUN);
				TFTimerSet(ADR(Timeout),3000+200,TRUE);
				TFTimerSet(ADR(Timer),3000,TRUE);
				TFCommandCase(ADR(CmdExe),1,CommandCase_INC);

			(* Case 1 - *)
			1: 
				TFCommandCase(ADR(CmdExe),10,CommandCase_JMP);

			(* Case 10 - Set automatico Soglie *)
			10:
				AspirazioneDX^.Command^.Aspirazione_ON_ScritturaSoglia 	:= TRUE;
				AspirazioneSX^.Command^.Aspirazione_ON_ScritturaSoglia 	:= TRUE;
				IF AspirazioneDX^.Status.CommandDone AND AspirazioneSX^.Status.CommandDone THEN
					AspirazioneDX^.Command^.Aspirazione_ON_ScritturaSoglia		:= FALSE;
					AspirazioneSX^.Command^.Aspirazione_ON_ScritturaSoglia		:= FALSE;
					TFCommandCase(ADR(CmdExe),100,CommandCase_JMP);
				ELSIF TFTimerDone(ADR(Timer)) THEN
					AspirazioneDX^.Command^.Aspirazione_ON_ScritturaSoglia		:= FALSE;
					AspirazioneSX^.Command^.Aspirazione_ON_ScritturaSoglia		:= FALSE;
					TFError(ErrTOHOME,ErrNULL,ADR(CmdExe),ADR(State),ADR(Error),ADR(ErrorLog));
				END_IF
			
	
			(* Case 100 *)
			100:TFStateUpdate(ADR(State),StateHOME_END);
				TFCommandExeClear(ADR(CmdExe));

			ELSE
				TFError(ErrNOCMDCASE,ErrNULL,ADR(CmdExe),ADR(State),ADR(Error),ADR(ErrorLog));
		END_CASE;
		
		IF AspirazioneDX^.Status.ErrorID <> ErrNULL THEN
			AspirazioneDX^.Command^.Aspirazione_ON_ScritturaSoglia 	:= TRUE;
			AspirazioneSX^.Command^.Aspirazione_ON_ScritturaSoglia 	:= TRUE;
			TFError(ErrCYLINDER,AspirazioneDX^.Status.ErrorID,ADR(CmdExe),ADR(State),ADR(Error),ADR(ErrorLog));
		ELSIF AspirazioneSX^.Status.ErrorID <> ErrNULL THEN
			AspirazioneDX^.Command^.Aspirazione_ON_ScritturaSoglia 	:= TRUE;
			AspirazioneSX^.Command^.Aspirazione_ON_ScritturaSoglia 	:= TRUE;
			TFError(ErrCYLINDER,AspirazioneSX^.Status.ErrorID,ADR(CmdExe),ADR(State),ADR(Error),ADR(ErrorLog));
		ELSIF TFTimerDone(ADR(Timeout)) THEN
			AspirazioneDX^.Command^.Aspirazione_ON_ScritturaSoglia 	:= TRUE;
			AspirazioneSX^.Command^.Aspirazione_ON_ScritturaSoglia 	:= TRUE;
			TFError(ErrCMDTIMEOUT,ErrNULL,ADR(CmdExe),ADR(State),ADR(Error),ADR(ErrorLog));
		END_IF

	(* ******************************************************************************************************** *)
	(* Manual *)
	(* ******************************************************************************************************** *)
	CmdMAN:
		CASE CmdExe.CmdCase OF
			(* Case 0 *)
			0: 	TFStateUpdate(ADR(State),StateMAN_RUN);
				TFTimerSet(ADR(Timeout),3000,TRUE);
				IF TFCommandParRead(CmdExe.Cmd.Parameter,ADR(ParametersArray),2) THEN
					MAN_Actuator	:= STRING_TO_UINT(ParametersArray.Parameters[0]);
					MAN_Cmd		:= STRING_TO_UINT(ParametersArray.Parameters[1]);
				ELSE
					TFError(ErrCMDPARNUM,ErrNULL,ADR(CmdExe),ADR(State),ADR(Error),ADR(ErrorLog));
					RETURN;
				END_IF;

				CASE MAN_Actuator OF
					(* Case 0..99 for Actuators *)
					(* Case 100..199  for Axis *)

					(* Case Nop *)
					0:	;

					(* Case 1: *)
					1:	CASE MAN_Cmd OF
							0:	;
							
							(* Case 10: Apertura Pinza *)
							10:	
								TFTimerSet(ADR(Timeout),30000,TRUE);
								TFCommandCase(ADR(CmdExe),10,CommandCase_JMP);
								
							(* Case 11: Chiusura Pinza *)
							11:	
								TFTimerSet(ADR(Timeout),30000,TRUE);
								TFCommandCase(ADR(CmdExe),10,CommandCase_JMP);

							(* Case 20: Sgancio Sblocco Rotazione *)
							20:	
								TFTimerSet(ADR(Timeout),3000,TRUE);
								TFCommandCase(ADR(CmdExe),20,CommandCase_JMP);
								
							(* Case 21: Aggancio Sblocco Rotazione *)
							21:	
								TFTimerSet(ADR(Timeout),3000,TRUE);
								TFCommandCase(ADR(CmdExe),20,CommandCase_JMP);

							(* Case 30: Ativazione Aspirazione Falda DX *)
							30:	
								TFTimerSet(ADR(Timeout),3000,TRUE);
								TFCommandCase(ADR(CmdExe),30,CommandCase_JMP);
								
							(* Case 31: Disattivazione Aspirazione Falda DX *)
							31:	
								TFTimerSet(ADR(Timeout),3000,TRUE);
								TFCommandCase(ADR(CmdExe),30,CommandCase_JMP);
								
							(* Case 40: Ativazione Aspirazione Falda SX *)
							40:	
								TFTimerSet(ADR(Timeout),3000,TRUE);
								TFCommandCase(ADR(CmdExe),40,CommandCase_JMP);
								
							(* Case 41: Disattivazione Aspirazione Falda SX *)
							41:	
								TFTimerSet(ADR(Timeout),3000,TRUE);
								TFCommandCase(ADR(CmdExe),40,CommandCase_JMP);

							(* Case 50: Ativazione Aspirazione SX *)
							50:	
								AspirazioneSX^.Command^.Aspirazione_ON 	:= TRUE;
								AspirazioneSX^.Command^.Aspirazione_OFF := FALSE;

								AspirazioneDX^.Command^.Aspirazione_ON 	:= TRUE;
								AspirazioneDX^.Command^.Aspirazione_OFF := FALSE;

								TFTimerSet(ADR(Timeout),3000,TRUE);
								TFCommandCase(ADR(CmdExe),50,CommandCase_JMP);
								
							(* Case 51: Disattivazione Aspirazione SX *)
							51:	
								AspirazioneSX^.Command^.Aspirazione_ON 	:= FALSE;
								AspirazioneSX^.Command^.Aspirazione_OFF := TRUE;
								TFTimerSet(ADR(Timeout),3000,TRUE);
								TFCommandCase(ADR(CmdExe),50,CommandCase_JMP);

							(* Case 60: Ativazione Aspirazione DX *)
							60:	
								AspirazioneDX^.Command^.Aspirazione_ON 	:= TRUE;
								AspirazioneDX^.Command^.Aspirazione_OFF := FALSE;
								TFTimerSet(ADR(Timeout),3000,TRUE);
								TFCommandCase(ADR(CmdExe),60,CommandCase_JMP);
								
							(* Case 61: Disattivazione Aspirazione SX *)
							61:	
								AspirazioneDX^.Command^.Aspirazione_ON 	:= FALSE;
								AspirazioneDX^.Command^.Aspirazione_OFF := TRUE;
								AspirazioneSX^.Command^.Aspirazione_ON 	:= FALSE;
								AspirazioneSX^.Command^.Aspirazione_OFF := TRUE;
								StatoPinza.ElementoPrelevato := FALSE;
								TFTimerSet(ADR(Timeout),3000,TRUE);
								TFCommandCase(ADR(CmdExe),60,CommandCase_JMP);
				
							(* Case 70: Ativazione Tastatori *)
							70:	
								TFTimerSet(ADR(Timeout),3000,TRUE);
								TFCommandCase(ADR(CmdExe),70,CommandCase_JMP);
								
							(* Case 71: Disattivazione Aspirazione SX *)
							71:	
								TFTimerSet(ADR(Timeout),3000,TRUE);
								TFCommandCase(ADR(CmdExe),70,CommandCase_JMP);

							ELSE
								TFError(ErrNOCMDCASE,ErrNULL,ADR(CmdExe),ADR(State),ADR(Error),ADR(ErrorLog));
						END_CASE;

					100:CASE MAN_Cmd OF
							0:	;
							ELSE
								TFError(ErrNOCMDCASE,ErrNULL,ADR(CmdExe),ADR(State),ADR(Error),ADR(ErrorLog));
						END_CASE;

					ELSE
						TFError(ErrNOCMDCASE,ErrNULL,ADR(CmdExe),ADR(State),ADR(Error),ADR(ErrorLog));
				END_CASE;

				//IF CmdExe.CmdCase = 0 THEN
					//TFCommandCase(ADR(CmdExe),1,CommandCase_INC);
				//END_IF

			(* Case 1 - *)
			1: 	IF (MAN_Cmd = 0) OR TFTimerDone(ADR(Timeout)) THEN
					(* Clear All Output Here *)
					;
					TFStateUpdate(ADR(State),StateMAN_END);
					TFCommandExeClear(ADR(CmdExe));
				END_IF;

			
			(* Case 10 - CilindroApertura *)
			10: ;

			(* Case 20 - CilindroSbloccoRotazione *)
			20: 
				;

			(* Case 30 - AspirazioneFaldaDX *)
			30: 
				;

			(* Case 40 - AspirazioneFaldaSX *)
			40: 
				;

			(* Case 50 - AspirazioneSX *)
			50: 
				IF AspirazioneSX^.Status.CommandDone AND AspirazioneDX^.Status.CommandDone THEN
					AspirazioneDX^.Command^.Aspirazione_ON 	:= FALSE;
					AspirazioneDX^.Command^.Aspirazione_OFF	:= FALSE;
					AspirazioneSX^.Command^.Aspirazione_ON 	:= FALSE;
					AspirazioneSX^.Command^.Aspirazione_OFF	:= FALSE;
					TFCommandCase(ADR(CmdExe),100,CommandCase_JMP);
				ELSIF AspirazioneSX^.Status.ErrorID <> ErrNULL THEN
					TFClearAllCmdModulePinza(AspirazioneDX,AspirazioneSX);
					TFError(ErrCYLINDER,AspirazioneSX^.Status.ErrorID,ADR(CmdExe),ADR(State),ADR(Error),ADR(ErrorLog));
				ELSIF AspirazioneDX^.Status.ErrorID <> ErrNULL THEN
					TFClearAllCmdModulePinza(AspirazioneDX,AspirazioneSX);
					TFError(ErrCYLINDER,AspirazioneDX^.Status.ErrorID,ADR(CmdExe),ADR(State),ADR(Error),ADR(ErrorLog));
				END_IF

			(* Case 60 - AspirazioneDX *)
			60: 
				IF AspirazioneSX^.Status.CommandDone AND AspirazioneDX^.Status.CommandDone THEN
					AspirazioneDX^.Command^.Aspirazione_ON 	:= FALSE;
					AspirazioneDX^.Command^.Aspirazione_OFF	:= FALSE;
					AspirazioneSX^.Command^.Aspirazione_ON 	:= FALSE;
					AspirazioneSX^.Command^.Aspirazione_OFF	:= FALSE;
					TFCommandCase(ADR(CmdExe),100,CommandCase_JMP);
				ELSIF AspirazioneSX^.Status.ErrorID <> ErrNULL THEN
					TFClearAllCmdModulePinza(AspirazioneDX,AspirazioneSX);
					TFError(ErrCYLINDER,AspirazioneSX^.Status.ErrorID,ADR(CmdExe),ADR(State),ADR(Error),ADR(ErrorLog));
				ELSIF AspirazioneDX^.Status.ErrorID <> ErrNULL THEN
					TFClearAllCmdModulePinza(AspirazioneDX,AspirazioneSX);
					TFError(ErrCYLINDER,AspirazioneDX^.Status.ErrorID,ADR(CmdExe),ADR(State),ADR(Error),ADR(ErrorLog));
				END_IF

			(* Case 70 - CilindroTasteggio *)
			70: 
				;
				
			(* Case 100 - End *)
			100:(* Clear All Output Here *)
				TFStateUpdate(ADR(State),StateMAN_END);
				TFCommandExeClear(ADR(CmdExe));

			ELSE
				TFError(ErrNOCMDCASE,ErrNULL,ADR(CmdExe),ADR(State),ADR(Error),ADR(ErrorLog));
		END_CASE;

		IF TFTimerDone(ADR(Timeout)) THEN
			TFClearAllCmdModulePinza(AspirazioneDX,AspirazioneSX);
			TFError(ErrCMDTIMEOUT,ErrNULL,ADR(CmdExe),ADR(State),ADR(Error),ADR(ErrorLog));
		END_IF
	

	(* ******************************************************************************************************** *)
	(* PRELOAD - Presa del pezzo *)
	(* ******************************************************************************************************** *)
	CmdPRELOAD:
		CASE CmdExe.CmdCase OF
			
			(* Case 0 - Init Command*)
			0: 	TFStateUpdate(ADR(State),StatePRELOAD_RUN);
				TFTimerSet(ADR(Timeout),30000+200,TRUE);
				TFTimerSet(ADR(Timer),30000,TRUE);
				PrelievoSuCavallina := FALSE;
				StatoPinza.ElementoPrelevato := FALSE;
				IF TFCommandParRead(CmdExe.Cmd.Parameter,ADR(ParametersArray),1) THEN
					PrelievoSuCavallina	:= STRING_TO_BOOL(ParametersArray.Parameters[0]);
					TFCommandCase(ADR(CmdExe),10,CommandCase_JMP);
				ELSE
					TFError(ErrCMDPARNUM,ErrNULL,ADR(CmdExe),ADR(State),ADR(Error),ADR(ErrorLog));
					RETURN;
				END_IF;
				
			(* Case 10 - CilindroApertura *)
			10: 
				TFCommandCase(ADR(CmdExe),40,CommandCase_JMP);
	
			(* Case 40 - AspirazioneDX + AspirazioneSX *)
			40: 
				AspirazioneDX^.Command^.Aspirazione_ON 	:= TRUE;
				AspirazioneDX^.Command^.Aspirazione_OFF := FALSE;
			
				AspirazioneSX^.Command^.Aspirazione_ON 	:= TRUE;
				AspirazioneSX^.Command^.Aspirazione_OFF := FALSE;
	
				IF AspirazioneDX^.Status.CommandDone AND AspirazioneSX^.Status.CommandDone THEN
					AspirazioneDX^.Command^.Aspirazione_ON 	:= FALSE;
					AspirazioneDX^.Command^.Aspirazione_OFF	:= FALSE;
					AspirazioneSX^.Command^.Aspirazione_ON 	:= FALSE;
					AspirazioneSX^.Command^.Aspirazione_OFF	:= FALSE;
					TFCommandCase(ADR(CmdExe),100,CommandCase_JMP);
				ELSIF AspirazioneSX^.Status.ErrorID <> ErrNULL THEN
					TFClearAllCmdModulePinza(AspirazioneDX,AspirazioneSX);
					TFError(ErrCYLINDER,AspirazioneSX^.Status.ErrorID,ADR(CmdExe),ADR(State),ADR(Error),ADR(ErrorLog));
				ELSIF AspirazioneDX^.Status.ErrorID <> ErrNULL THEN
					TFClearAllCmdModulePinza(AspirazioneDX,AspirazioneSX);
					TFError(ErrCYLINDER,AspirazioneDX^.Status.ErrorID,ADR(CmdExe),ADR(State),ADR(Error),ADR(ErrorLog));
				END_IF
				
			(* Case 100 *)
			100:TFStateUpdate(ADR(State),StatePRELOAD_END);
				TFCommandExeClear(ADR(CmdExe));

			ELSE
				TFError(ErrNOCMDCASE,ErrNULL,ADR(CmdExe),ADR(State),ADR(Error),ADR(ErrorLog));
		END_CASE

		IF TFTimerDone(ADR(Timeout)) THEN
			TFClearAllCmdModulePinza(AspirazioneDX,AspirazioneSX);
			TFError(ErrCMDTIMEOUT,ErrNULL,ADR(CmdExe),ADR(State),ADR(Error),ADR(ErrorLog));
		END_IF
	


	(* ******************************************************************************************************** *)
	(* LOAD - Presa del pezzo *)
	(* ******************************************************************************************************** *)
	CmdCHECKPRESENCE:
		CASE CmdExe.CmdCase OF
			
			(* Case 0 - Init Command*)
			0: 	TFStateUpdate(ADR(State),StateCHECKPRESENCE_RUN);
				TFTimerSet(ADR(Timeout),60000.0+100+HMI_TempoControlloPresaPiastrella,TRUE);
				TFTimerSet(ADR(Timer),2000.0+HMI_TempoControlloPresaPiastrella,TRUE);
				TFTimerSet(ADR(TimerPresaPiastrella),HMI_TempoControlloPresaPiastrella,TRUE);
				StatoPinza.ElementoPrelevato := FALSE;

				TFCommandCase(ADR(CmdExe),1,CommandCase_INC);
				
			(* Case 1 - *)					
			1:
				IF IN.ByPassSensoreVuoto THEN
					StatoPinza.ElementoPrelevato := TRUE;
				ELSE
					StatoPinza.ElementoPrelevato := FALSE;
				END_IF

				IF IN.ByPassSensoreVuoto OR TFTimerDone(ADR(TimerPresaPiastrella)) THEN 
					//Tutte piastrelle o tutte falde
					IF (AspirazioneDX^.Status.DepressioneSoglia1_OK AND AspirazioneSX^.Status.DepressioneSoglia1_OK) OR IN.ByPassSensoreVuoto THEN
						StatoPinza.ElementoPrelevato := TRUE;
						TFCommandCase(ADR(CmdExe),100,CommandCase_JMP);					
					ELSIF TFTimerDone(ADR(TimerPresaPiastrella)) THEN
						TFCommandCase(ADR(CmdExe),100,CommandCase_JMP);
						StatoPinza.ElementoPrelevato := FALSE;	
					END_IF			
				ELSIF TFTimerDone(ADR(TimerPresaPiastrella)) THEN
					TFCommandCase(ADR(CmdExe),100,CommandCase_JMP);
					StatoPinza.ElementoPrelevato := FALSE;
				END_IF			
				IF TFTimerDone(ADR(Timer)) THEN
					TFClearAllCmdModulePinza(AspirazioneDX,AspirazioneSX);
					TFError(ErrMalfunzionamentoSensoriPresenzaPinza,ErrNULL,ADR(CmdExe),ADR(State),ADR(Error),ADR(ErrorLog));
				ELSIF TFTimerDone(ADR(Timeout)) THEN
					TFClearAllCmdModulePinza(AspirazioneDX,AspirazioneSX);
					TFError(ErrCMDTIMEOUT,ErrNULL,ADR(CmdExe),ADR(State),ADR(Error),ADR(ErrorLog));
				END_IF
							
			(* Case 100 *)
			100:TFStateUpdate(ADR(State),StateCHECKPRESENCE_END);
				TFCommandExeClear(ADR(CmdExe));

			ELSE
				TFError(ErrNOCMDCASE,ErrNULL,ADR(CmdExe),ADR(State),ADR(Error),ADR(ErrorLog));
		END_CASE
		
	
	(* ******************************************************************************************************** *)
	(* UNLOAD - Attivazione aspirazione + discesa ventose *)
	(* ******************************************************************************************************** *)
	CmdUNLOAD:
		CASE CmdExe.CmdCase OF
			
			(* Case 0 - Init Command*)
			0: 	TFStateUpdate(ADR(State),StateUNLOAD_RUN);
				TFTimerSet(ADR(Timeout),30000+200,TRUE);
				TFTimerSet(ADR(Timer),30000,TRUE);
				StatoPinza.ElementoPrelevato := FALSE;
				TFCommandCase(ADR(CmdExe),20,CommandCase_JMP);				
				
				
		
			(* Case 20 - Disattivazione aspirazione piastrella *)		
			20: 
				AspirazioneDX^.Command^.Aspirazione_ON 	:= FALSE;
				AspirazioneDX^.Command^.Aspirazione_OFF := TRUE;
			
				AspirazioneSX^.Command^.Aspirazione_ON 	:= FALSE;
				AspirazioneSX^.Command^.Aspirazione_OFF := TRUE;
		
				IF AspirazioneDX^.Status.CommandDone AND AspirazioneSX^.Status.CommandDone THEN
					AspirazioneDX^.Command^.Aspirazione_ON 	:= FALSE;
					AspirazioneDX^.Command^.Aspirazione_OFF	:= FALSE;
					AspirazioneSX^.Command^.Aspirazione_ON 	:= FALSE;
					AspirazioneSX^.Command^.Aspirazione_OFF	:= FALSE;
					TFTimerSet(ADR(TimerAspirazione),HMI_TempoRilascioInDeposito,TRUE);
					TFCommandCase(ADR(CmdExe),30,CommandCase_JMP);
				ELSIF AspirazioneSX^.Status.ErrorID <> ErrNULL THEN
					TFClearAllCmdModulePinza(AspirazioneDX,AspirazioneSX);
					TFError(ErrCYLINDER,AspirazioneSX^.Status.ErrorID,ADR(CmdExe),ADR(State),ADR(Error),ADR(ErrorLog));
				ELSIF AspirazioneDX^.Status.ErrorID <> ErrNULL THEN
					TFClearAllCmdModulePinza(AspirazioneDX,AspirazioneSX);
					TFError(ErrCYLINDER,AspirazioneDX^.Status.ErrorID,ADR(CmdExe),ADR(State),ADR(Error),ADR(ErrorLog));
				END_IF
			
			(* Case 30 - Attesa tempo distacco *)		
			30:
				IF TFTimerDone(ADR(TimerAspirazione)) THEN
					IF IN.RichiestaRicalibrazioneOvemEsterna THEN
						IN.RichiestaRicalibrazioneOvemEsterna := FALSE;
						TFCommandCase(ADR(CmdExe),40,CommandCase_JMP);
					ELSE
						TFCommandCase(ADR(CmdExe),100,CommandCase_JMP);
					END_IF		
				END_IF
				
			(* Case 40 - Attesa tempo distacco *)		
			40:	
				AspirazioneDX^.Command^.Aspirazione_ON_ScritturaSoglia 	:= TRUE;
				AspirazioneSX^.Command^.Aspirazione_ON_ScritturaSoglia 	:= TRUE;
				IF AspirazioneDX^.Status.CommandDone AND AspirazioneSX^.Status.CommandDone THEN
					AspirazioneDX^.Command^.Aspirazione_ON_ScritturaSoglia		:= FALSE;
					AspirazioneSX^.Command^.Aspirazione_ON_ScritturaSoglia		:= FALSE;
					TFCommandCase(ADR(CmdExe),100,CommandCase_JMP);
				ELSIF TFTimerDone(ADR(Timer)) THEN
					AspirazioneDX^.Command^.Aspirazione_ON_ScritturaSoglia		:= FALSE;
					AspirazioneSX^.Command^.Aspirazione_ON_ScritturaSoglia		:= FALSE;
					TFError(ErrTOHOME,ErrNULL,ADR(CmdExe),ADR(State),ADR(Error),ADR(ErrorLog));
				END_IF
				
		
			(* Case 100 *)
			100:TFStateUpdate(ADR(State),StateUNLOAD_END);
				TFCommandExeClear(ADR(CmdExe));

			ELSE
				TFError(ErrNOCMDCASE,ErrNULL,ADR(CmdExe),ADR(State),ADR(Error),ADR(ErrorLog));
		END_CASE

		IF TFTimerDone(ADR(Timeout)) THEN
			TFClearAllCmdModulePinza(AspirazioneDX,AspirazioneSX);
			TFError(ErrCMDTIMEOUT,ErrNULL,ADR(CmdExe),ADR(State),ADR(Error),ADR(ErrorLog));
		END_IF


	ELSE
		TFError(ErrNOCMD,ErrNULL,ADR(CmdExe),ADR(State),ADR(Error),ADR(ErrorLog));

END_CASE;


(* ******************************************************************************************************** *)
(* State Input/Output *)
(* ******************************************************************************************************** *)
(* Fill Input/Output bit with sensor, electrovalve, etc. status *)

StatoPinza.LatoDxPiastrellaInPresa	:= (AspirazioneDX^.Status.DepressioneSoglia1_OK  OR (IN.ByPassSensoreVuoto AND StatoPinza.ElementoPrelevato));
StatoPinza.LatoSxPiastrellaInPresa	:=(AspirazioneSX^.Status.DepressioneSoglia1_OK  OR (IN.ByPassSensoreVuoto AND StatoPinza.ElementoPrelevato));

(* ******************************************************************************************************** *)
(* Input *)
(* ******************************************************************************************************** *)

(* ******************************************************************************************************** *)
(* Alarm *)
(* ******************************************************************************************************** *)

(* ******************************************************************************************************** *)
(* Error Check - Clear All Output!!! *)
(* ******************************************************************************************************** *)
IF Error.Code > ErrNULL THEN
	IF CmdExe.Code <> CmdNOP THEN
		IF CmdExe.Code <> CmdSTOP AND
			CmdExe.Code <> CmdPOWER AND
			CmdExe.Code <> CmdRESET AND
			CmdExe.Code <> CmdMAN AND
			CmdExe.Code <> CmdLOAD AND
			CmdExe.Code <> CmdUNLOAD THEN
			TFCommandClear(ADR(CmdNext));
			TFCommandExeClear(ADR(CmdExe));

			(* Clear All Output Here *)

		END_IF;
	END_IF;
END_IF;


(* ******************************************************************************************************** *)
(* Common Outputs *)
(* ******************************************************************************************************** *)

END_FUNCTION_BLOCK

// ---- POUs/TFModules/Utility/TFClearAllCmdModulePinza.TcPOU
FUNCTION TFClearAllCmdModulePinza : bool
VAR_INPUT
	AspirazioneDX : POINTER TO TF_VacumOVEM;
	AspirazioneSX : POINTER TO TF_VacumOVEM;
END_VAR
VAR
END_VAR

TFOVEMClearAllCommand(AspirazioneDX^.Command);
TFOVEMClearAllCommand(AspirazioneSX^.Command);

END_FUNCTION

// ---- POUs/TFModules/Utility/TFCylinder_HasCommand.TcPOU
FUNCTION TFCylinder_HasCommand : bool
VAR_INPUT
	Command: CylinderCommand;
END_VAR
VAR
END_VAR

Cylinder_HasCommand:=
Command.Deactivation OR 
Command.Activation OR 
Command.Hold OR
Command.Abort;

END_FUNCTION

// ---- POUs/TFPalletizerDataTF/FunzionePerNuovaGestioneTrasporti/TFPackCodePresenteInZona_old.TcPOU
FUNCTION TFPackCodePresenteInZona_old : INT
VAR_INPUT
	//HandlingPackTable : POINTER TO TFHandlingPackTable;
	ArrayPacchi : POINTER TO DUT_ArrayPacchi;
	WorkAreaZone : POINTER TO TFMachinePalletizer_WorkAreaZone;
	WorkArea : INT;
END_VAR
VAR
	w : INT;
	n : INT;
	i : INT;
	a : INT;
END_VAR

TFPackCodePresenteInZona := 0; 

//FOR w:=1 TO MAXDIMARRAYPACCHI DO
	IF ArrayPacchi^.Pacco[1].PC > 0 THEN
		FOR n:=1 TO MAXZONE DO
			FOR a:=1 TO MAXAREA DO
				IF WorkAreaZone^.Zone[n].WorkArea[a] = WorkArea THEN
					FOR i:=1 TO MAXFORMINGCODE DO
						(* Verifico se il Pacco presente nel WPP è destinato ad una Zona *)
						IF WorkAreaZone^.Zone[n].Code[i] = ArrayPacchi^.Pacco[1].PC THEN
							TFPackCodePresenteInZona := ArrayPacchi^.Pacco[w].PC;
							RETURN;
						END_IF
					END_FOR
				END_IF
			END_FOR
		END_FOR
	END_IF
//END_FOR

END_FUNCTION

// ---- POUs/TFPalletizerDataTF/NON_USATE/TFCalcoliFuoriIngombriColonne.TcPOU
FUNCTION_BLOCK TFCalcoliFuoriIngombriColonne
VAR_INPUT
	Traiettoria : POINTER TO TFTraiettoria;
	WorkSpace : POINTER TO TFMachinePalletizer_WorkSpace;
	WorkFootprint : POINTER TO ARRAY [1..MAXFOOTPRINT] OF TFMachinePalletizer_WorkFootprint; //Ingombri
	WorkPickPoint : POINTER TO ARRAY [1..MAXPICKPOINT] OF TFMachinePalletizer_WorkPickPoint;
	//WorkPickPointState : POINTER TO ARRAY [1..MAXPICKPOINT] OF TFMachinePalletizer_WorkPickPointState;
	WorkArea : POINTER TO ARRAY [1..MAXAREA] OF TFMachinePalletizer_WorkArea;
	WorkAreaState : POINTER TO ARRAY [1..MAXAREA] OF TFMachinePalletizer_WorkAreaState;
	Pallet : POINTER TO ARRAY [1..MAXPALLET] OF TFMachinePalletizer_Pallet;
	Layer : POINTER TO ARRAY [1..MAXLAYER] OF TFMachinePalletizer_Layer;
	Forming : POINTER TO ARRAY [1..MAXFORMING] OF TFMachinePalletizer_FormingForSlab;
	PickPlaceParameters	: POINTER TO TFMachinePalletizer_ParametersFromHMI;
	Mission : POINTER TO TFMachinePalletizer_Mission;
	
	WorkAreaManager : POINTER TO TFWorkAreaManager;
	ModuleAX_X : POINTER TO TFModulePalletizer_Ax;
	ModuleAX_Y : POINTER TO TFModulePalletizer_Ax;
	ModuleAX_Z : POINTER TO TFModulePalletizer_Ax;
	ModuleAX_J : POINTER TO TFModulePalletizer_Ax;
	ModuleAX_K : POINTER TO TFModulePalletizer_Ax;
	AbilitaCalcoloIngombroOttimizzato : BOOL := TRUE; //Abilitazione dell'utilizzo degli ingombri ottimizzati... calcoli in base all'angolo di rotazione della pinza
END_VAR
VAR
	f : INT;
	a : INT;
	P : INT;
	wa : int;
	waDXSX : INT;
	AltezzaDiIngombroArea : REAL;
	AltezzaDiIngombroOstacoli : REAL;
	AltezzaDiIngombroPuntiPrelievo : REAL;
	AssegnaQuote : BOOL;
	
	LunghezzaMAX 	: LREAL;//LunghezzaMAX Totale pinza
	LarghezzaMAX 	: LREAL;//Larghezza Totale pinza
	SpessoreMAX  	: LREAL;//Spessore Totale pinza

	IngombroX_Pos : LREAL;//Ingombro della pinza nella Metà POSITIVA della pinza lungo X
	IngombroY_Pos : LREAL;//Ingombro della pinza nella Metà POSITIVA della pinza lungo Y
	
	IngombroX_Neg : LREAL;//Ingombro della pinza nella Metà NEGATIVA della pinza lungo X
	IngombroY_Neg : LREAL;//Ingombro della pinza nella Metà NEGATIVA della pinza lungo Y
	
	IngombroZ : LREAL;//Ingombro della pinza lungo Z
	
	IngombroVerticalePinzaMAX : REAL;
	IngombroVerticaleMaxElementi : REAL;
	//DirezioneXPositiva_Dep : BOOL;
	//DirezioneXNegativa_Dep : BOOL;
	//DirezioneXPositiva_Prel : BOOL;
	//DirezioneXNegativa_Prel : BOOL;
	DirezioneZPositiva : BOOL;
	DirezioneZNegativa : BOOL;
	DirezioneXNegativa : BOOL;
	DirezioneXPositiva : BOOL;
	
	
	WASX : UINT;
	WADX : UINT;
	WAPARTENZA : UINT;
	WADESTINAZIONE : UINT;
	LarghezzaPickPoint : REAL;
	
	
	FuoriIngombroYNecessarioTMP : BOOL;
	QuotaX_ConsensoRotazionePinza_RaggiuntaTMP : BOOL;
	ConsensoTraslazioneY_TraColonneTMP : BOOL;
	AsseXInFinestraDiPrelievoPaccoTMP : BOOL;
	AsseJInFinestraDiPrelievoPaccoTMP : BOOL;
	
	OffsetSicurezza_Y : real := 80;
	
	
	Pinza_InIngombroColonne_Partenza: BOOL; //Indica che la posizione della pinza è in ingombro colonne alla partenza del ciclo/ REAL TIME
	IngombroOttimizzatoY_Destinazione: LREAL;
	IngombroOttimizzatoX_Destinazione: LREAL;
	IngombroOttimizzatoX_InPuntoDiPrelievo: LREAL;
	IngombroOttimizzatoY_InPuntoDiPrelievo: LREAL;
	IngombroOttimizzatoY_InPuntoDiDeposito: LREAL;
	IngombroOttimizzatoX_InPuntoDiDeposito: LREAL;
	//Pinza_InIngombroColonne_Attuale: BOOL;
	//Pinza_InIngombroColonne_Destinazione: BOOL;
	AsseJInFinestraDiPrelievoPallet: BOOL;
	AsseXInFinestraDiPrelievoPallet: BOOL;
	AsseYInFinestraDiPrelievoPallet: BOOL;
	AsseXInFinestraDiRiposo: BOOL;
	AsseYInFinestraDiRiposo: BOOL;
	AsseJInFinestraDiRiposo: BOOL;
	AsseXInFinestraDiDestinazione: BOOL;
	AsseJInFinestraDiDestinazione: BOOL;
	AsseYInFinestraDiDestinazione: BOOL;
	IngombroOttimizzatoX_InTransito: LREAL;
	IngombroOttimizzatoY_InTransito: LREAL;
	Pinza_InIngombroColonne_Transito: BOOL;
	Angolo: INT;
	CalcolaIngombro: BOOL;
	AsseXInFinestraDiPrelievo: BOOL;
	AsseYInFinestraDiPrelievo: BOOL;
	AsseJInFinestraDiPrelievo: BOOL;
	
	QuotaFuoriIngombro_Attuale_Y 		: LREAL;
	QuotaFuoriIngombro_Prelievo_Y 		: LREAL;
	QuotaFuoriIngombro_Deposito_Y		: LREAL;
	
	TFCalcolaQuotaIngombroColonne : TFCalcolaQuotaIngombroColonne;
	TFCalcoloIngombroOttimizzatoPinza : TFCalcoloIngombroOttimizzatoPinza;
	QuotaFuoriIngombro_Destinazione_Y: LREAL;
	WorkAreaManagerState_OLD: INT;
END_VAR

(* Calcolo delle dimensioni della pinza in base al tipo di ciclo in corso *)
CASE WorkAreaManager^.State OF
	WAMANAGER_NOP,
	
	WAMANAGER_CICLO_RIPOSO_INIT,
		
	WAMANAGER_CICLO_RIPOSO_RUN:
		
		SpessoreMAX 	:= Dimensioni_Pinza.Spessore;
		LunghezzaMAX 	:= Dimensioni_Pinza.Lunghezza;
		LarghezzaMAX    := Dimensioni_Pinza.Larghezza;
						
		IngombroX_Pos 	:=  LunghezzaMAX/2;
		IngombroX_Neg 	:=  LunghezzaMAX/2;

		IngombroY_Pos 	:= ABS(LarghezzaMAX/2 * COS(deg_to_rad(90+ModuleAX_J^.Ax^.AxRef^.NcToPlc.ActPos)) +
							SpessoreMAX * SIN(deg_to_rad(90+ModuleAX_J^.Ax^.AxRef^.NcToPlc.ActPos)));
							
		IngombroY_Neg 	:= ABS(LarghezzaMAX/2 * COS(deg_to_rad(90+ModuleAX_J^.Ax^.AxRef^.NcToPlc.ActPos)) -
							SpessoreMAX * SIN(deg_to_rad(90+ModuleAX_J^.Ax^.AxRef^.NcToPlc.ActPos)));	

		IngombroZ		:= Dimensioni_Pinza.Larghezza/2 * SIN(deg_to_rad(90+ModuleAX_J^.Ax^.AxRef^.NcToPlc.ActPos)) +
							SpessoreMAX * COS(deg_to_rad(90+ModuleAX_J^.Ax^.AxRef^.NcToPlc.ActPos));		
									
	WAMANAGER_CICLO_PRELIEVO_FALDA_RUN:
	
		SpessoreMAX 	:= Dimensioni_Pinza.Spessore;
		LunghezzaMAX 	:= Dimensioni_Pinza.Lunghezza;
		LarghezzaMAX    := Dimensioni_Pinza.Larghezza;
						
		IngombroX_Pos 	:=  LunghezzaMAX/2;
		IngombroX_Neg 	:=  LunghezzaMAX/2;

		IngombroY_Pos 	:= ABS(LarghezzaMAX/2 * COS(deg_to_rad(90+ModuleAX_J^.Ax^.AxRef^.NcToPlc.ActPos)) +
							SpessoreMAX * SIN(deg_to_rad(90+ModuleAX_J^.Ax^.AxRef^.NcToPlc.ActPos)));
							
		IngombroY_Neg 	:= ABS(LarghezzaMAX/2 * COS(deg_to_rad(90+ModuleAX_J^.Ax^.AxRef^.NcToPlc.ActPos)) -
							SpessoreMAX * SIN(deg_to_rad(90+ModuleAX_J^.Ax^.AxRef^.NcToPlc.ActPos)));	

		IngombroZ		:= Dimensioni_Pinza.Larghezza/2 * SIN(deg_to_rad(90+ModuleAX_J^.Ax^.AxRef^.NcToPlc.ActPos)) +
							SpessoreMAX * COS(deg_to_rad(90+ModuleAX_J^.Ax^.AxRef^.NcToPlc.ActPos));

	WAMANAGER_CICLO_DEPOSITO_FALDA_RUN:
		
		SpessoreMAX 	:= Dimensioni_Pinza.Spessore;
		LunghezzaMAX 	:= MAX(Dimensioni_Pinza.Lunghezza,Mission^.XDim);
		LarghezzaMAX    := MAX(Dimensioni_Pinza.Larghezza,Mission^.YDim);
						
		IngombroX_Pos 	:=  LunghezzaMAX/2;
		IngombroX_Neg 	:=  LunghezzaMAX/2;

		IngombroY_Pos 	:= ABS(LarghezzaMAX/2 * COS(deg_to_rad(90+ModuleAX_J^.Ax^.AxRef^.NcToPlc.ActPos)) +
							SpessoreMAX * SIN(deg_to_rad(90+ModuleAX_J^.Ax^.AxRef^.NcToPlc.ActPos)));
							
		IngombroY_Neg 	:= ABS(LarghezzaMAX/2 * COS(deg_to_rad(90+ModuleAX_J^.Ax^.AxRef^.NcToPlc.ActPos)) -
							SpessoreMAX * SIN(deg_to_rad(90+ModuleAX_J^.Ax^.AxRef^.NcToPlc.ActPos)));	

		IngombroZ		:= Dimensioni_Pinza.Larghezza/2 * SIN(deg_to_rad(90+ModuleAX_J^.Ax^.AxRef^.NcToPlc.ActPos)) +
							SpessoreMAX * COS(deg_to_rad(90+ModuleAX_J^.Ax^.AxRef^.NcToPlc.ActPos));		
									
				
	WAMANAGER_CICLO_PRELIEVO_LASTRA_WA_RUN:
	
		SpessoreMAX 	:= Dimensioni_Pinza.Spessore;
		LunghezzaMAX 	:= Dimensioni_Pinza.Lunghezza;
		LarghezzaMAX    := Dimensioni_Pinza.Larghezza;
						
		IngombroX_Pos 	:=  LunghezzaMAX/2;
		IngombroX_Neg 	:=  LunghezzaMAX/2;

		IngombroY_Pos 	:= ABS(LarghezzaMAX/2 * COS(deg_to_rad(90+ModuleAX_J^.Ax^.AxRef^.NcToPlc.ActPos)) +
							SpessoreMAX * SIN(deg_to_rad(90+ModuleAX_J^.Ax^.AxRef^.NcToPlc.ActPos)));
							
		IngombroY_Neg 	:= ABS(LarghezzaMAX/2 * COS(deg_to_rad(90+ModuleAX_J^.Ax^.AxRef^.NcToPlc.ActPos)) -
							SpessoreMAX * SIN(deg_to_rad(90+ModuleAX_J^.Ax^.AxRef^.NcToPlc.ActPos)));	

		IngombroZ		:= Dimensioni_Pinza.Larghezza/2 * SIN(deg_to_rad(90+ModuleAX_J^.Ax^.AxRef^.NcToPlc.ActPos)) +
							SpessoreMAX * COS(deg_to_rad(90+ModuleAX_J^.Ax^.AxRef^.NcToPlc.ActPos));
					
	WAMANAGER_CICLO_DEPOSITO_LASTRA_SU_PAREGGIATORE_RUN:
	
		SpessoreMAX 	:= Dimensioni_Pinza.Spessore;
		LunghezzaMAX 	:= MAX(Dimensioni_Pinza.Lunghezza,Mission^.XDim);
		LarghezzaMAX    := MAX(Dimensioni_Pinza.Larghezza,Mission^.YDim);
						
		IngombroX_Pos 	:=  LunghezzaMAX/2;
		IngombroX_Neg 	:=  LunghezzaMAX/2;

		IngombroY_Pos 	:= ABS(LarghezzaMAX/2 * COS(deg_to_rad(90+ModuleAX_J^.Ax^.AxRef^.NcToPlc.ActPos)) +
							SpessoreMAX * SIN(deg_to_rad(90+ModuleAX_J^.Ax^.AxRef^.NcToPlc.ActPos)));
							
		IngombroY_Neg 	:= ABS(LarghezzaMAX/2 * COS(deg_to_rad(90+ModuleAX_J^.Ax^.AxRef^.NcToPlc.ActPos)) -
							SpessoreMAX * SIN(deg_to_rad(90+ModuleAX_J^.Ax^.AxRef^.NcToPlc.ActPos)));	

		IngombroZ		:= Dimensioni_Pinza.Larghezza/2 * SIN(deg_to_rad(90+ModuleAX_J^.Ax^.AxRef^.NcToPlc.ActPos)) +
							SpessoreMAX * COS(deg_to_rad(90+ModuleAX_J^.Ax^.AxRef^.NcToPlc.ActPos));
					
	WAMANAGER_CICLO_PRELIEVO_LASTRA_DA_PAREGGIATORE_RUN:
	
		SpessoreMAX 	:= Dimensioni_Pinza.Spessore;
		LunghezzaMAX 	:= Dimensioni_Pinza.Lunghezza;
		LarghezzaMAX    := Dimensioni_Pinza.Larghezza;
						
		IngombroX_Pos 	:=  LunghezzaMAX/2;
		IngombroX_Neg 	:=  LunghezzaMAX/2;

		IngombroY_Pos 	:= ABS(LarghezzaMAX/2 * COS(deg_to_rad(90+ModuleAX_J^.Ax^.AxRef^.NcToPlc.ActPos)) +
							SpessoreMAX * SIN(deg_to_rad(90+ModuleAX_J^.Ax^.AxRef^.NcToPlc.ActPos)));
							
		IngombroY_Neg 	:= ABS(LarghezzaMAX/2 * COS(deg_to_rad(90+ModuleAX_J^.Ax^.AxRef^.NcToPlc.ActPos)) -
							SpessoreMAX * SIN(deg_to_rad(90+ModuleAX_J^.Ax^.AxRef^.NcToPlc.ActPos)));	

		IngombroZ		:= Dimensioni_Pinza.Larghezza/2 * SIN(deg_to_rad(90+ModuleAX_J^.Ax^.AxRef^.NcToPlc.ActPos)) +
							SpessoreMAX * COS(deg_to_rad(90+ModuleAX_J^.Ax^.AxRef^.NcToPlc.ActPos));				
					
	WAMANAGER_CICLO_DEPOSITO_LASTRA_WA_RUN:
	
		SpessoreMAX 	:= Dimensioni_Pinza.Spessore;
		LunghezzaMAX 	:= MAX(Dimensioni_Pinza.Lunghezza,Mission^.XDim);
		LarghezzaMAX    := MAX(Dimensioni_Pinza.Larghezza,Mission^.YDim);
						
		IngombroX_Pos 	:=  LunghezzaMAX/2;
		IngombroX_Neg 	:=  LunghezzaMAX/2;

		IngombroY_Pos 	:= ABS(LarghezzaMAX/2 * COS(deg_to_rad(90+ModuleAX_J^.Ax^.AxRef^.NcToPlc.ActPos)) +
							SpessoreMAX * SIN(deg_to_rad(90+ModuleAX_J^.Ax^.AxRef^.NcToPlc.ActPos)));
							
		IngombroY_Neg 	:= ABS(LarghezzaMAX/2 * COS(deg_to_rad(90+ModuleAX_J^.Ax^.AxRef^.NcToPlc.ActPos)) -
							SpessoreMAX * SIN(deg_to_rad(90+ModuleAX_J^.Ax^.AxRef^.NcToPlc.ActPos)));	

		IngombroZ		:= Dimensioni_Pinza.Larghezza/2 * SIN(deg_to_rad(90+ModuleAX_J^.Ax^.AxRef^.NcToPlc.ActPos)) +
							SpessoreMAX * COS(deg_to_rad(90+ModuleAX_J^.Ax^.AxRef^.NcToPlc.ActPos));

	WAMANAGER_CICLO_PRELIEVO_LASTRA_PP_RUN:
	
		SpessoreMAX 	:= Dimensioni_Pinza.Spessore;
		LunghezzaMAX 	:= Dimensioni_Pinza.Lunghezza;
		LarghezzaMAX    := Dimensioni_Pinza.Larghezza;
						
		IngombroX_Pos 	:=  LunghezzaMAX/2;
		IngombroX_Neg 	:=  LunghezzaMAX/2;

		IngombroY_Pos 	:= ABS(LarghezzaMAX/2 * COS(deg_to_rad(90+ModuleAX_J^.Ax^.AxRef^.NcToPlc.ActPos)) +
							SpessoreMAX * SIN(deg_to_rad(90+ModuleAX_J^.Ax^.AxRef^.NcToPlc.ActPos)));
							
		IngombroY_Neg 	:= ABS(LarghezzaMAX/2 * COS(deg_to_rad(90+ModuleAX_J^.Ax^.AxRef^.NcToPlc.ActPos)) -
							SpessoreMAX * SIN(deg_to_rad(90+ModuleAX_J^.Ax^.AxRef^.NcToPlc.ActPos)));	

		IngombroZ		:= Dimensioni_Pinza.Larghezza/2 * SIN(deg_to_rad(90+ModuleAX_J^.Ax^.AxRef^.NcToPlc.ActPos)) +
							SpessoreMAX * COS(deg_to_rad(90+ModuleAX_J^.Ax^.AxRef^.NcToPlc.ActPos));			

	WAMANAGER_CICLO_DEPOSITO_LASTRA_PP_RUN:
	
		SpessoreMAX 	:= Dimensioni_Pinza.Spessore;
		LunghezzaMAX 	:= MAX(Dimensioni_Pinza.Lunghezza,Mission^.XDim);
		LarghezzaMAX    := MAX(Dimensioni_Pinza.Larghezza,Mission^.YDim);
						
		IngombroX_Pos 	:=  LunghezzaMAX/2;
		IngombroX_Neg 	:=  LunghezzaMAX/2;

		IngombroY_Pos 	:= ABS(LarghezzaMAX/2 * COS(deg_to_rad(90+ModuleAX_J^.Ax^.AxRef^.NcToPlc.ActPos)) +
							SpessoreMAX * SIN(deg_to_rad(90+ModuleAX_J^.Ax^.AxRef^.NcToPlc.ActPos)));
							
		IngombroY_Neg 	:= ABS(LarghezzaMAX/2 * COS(deg_to_rad(90+ModuleAX_J^.Ax^.AxRef^.NcToPlc.ActPos)) -
							SpessoreMAX * SIN(deg_to_rad(90+ModuleAX_J^.Ax^.AxRef^.NcToPlc.ActPos)));	

		IngombroZ		:= Dimensioni_Pinza.Larghezza/2 * SIN(deg_to_rad(90+ModuleAX_J^.Ax^.AxRef^.NcToPlc.ActPos)) +
							SpessoreMAX * COS(deg_to_rad(90+ModuleAX_J^.Ax^.AxRef^.NcToPlc.ActPos));						
	
END_CASE
(**********************************************************************************************)
(**********************************************************************************************)
(* Setto la variabile per eseguire i calcoli al cambio del WAMANAGER *)
IF WorkAreaManager^.State <> WorkAreaManagerState_OLD THEN
	WorkAreaManagerState_OLD := WorkAreaManager^.State;
	CalcolaIngombro := TRUE; 
END_IF

CASE WorkAreaManager^.State OF
	WAMANAGER_NOP:;
	
	WAMANAGER_CICLO_RIPOSO_INIT:;
		
	WAMANAGER_CICLO_RIPOSO_RUN:
	
		DirezioneXPositiva := TFDirezioneAssePositiva(Posizione_Attuale:=ModuleAX_X^.Ax^.Status.ActPosition,Posizione_Finale:=Mission^.XPick);
		DirezioneXNegativa := NOT DirezioneXPositiva;
		(* Valuto se con l'asse X sono fuori dall'area delle colonne *)
		QuotaX_ConsensoRotazionePinza_Raggiunta := TFPinzaInFuoriIngombroColonne_DirezioneX(DirezioneXPositiva:=DirezioneXPositiva,
																							AsseInMoto:=ModuleAX_X^.Ax^.AxRef^.Status.Moving,
																							PosizioneAttuale:=ModuleAX_X^.Ax^.Status.ActPosition,
																							PosizioneColonna_X:=WorkFootprint^[5].X,  
																							IngombroColonna_X:=WorkFootprint^[5].XDim,
																							IngombroX_Pos:=IngombroX_Pos,
																							IngombroX_Neg:=IngombroX_Neg);
		IF CalcolaIngombro THEN
			CalcolaIngombro := FALSE;
			(* Definisco il tipo di area in cui si trova a lavorare il pallettizzatore *)
			AreaInLavoroPositiva := FALSE;
			AreaInLavoroNegativa := FALSE;
			AreaInLavoroPositivaNegativa := TRUE; 
									
			(**************************************************************************************************************************************************)
			(* Valuto la direzione della X *)
			(**************************************************************************************************************************************************)
			DirezioneXPositiva := TFDirezioneAssePositiva(Posizione_Attuale:=ModuleAX_X^.Ax^.Status.ActPosition,Posizione_Finale:=Mission^.XPick);
			DirezioneXNegativa := NOT DirezioneXPositiva;
			
			(**************************************************************************************************************************************************)
			(* Valuto la direzione della X *)
			(**************************************************************************************************************************************************)
						
			(**************************************************************************************************************************************************)
			(* Ingombro MASSIMO della pinza durante il transito *)
			(**************************************************************************************************************************************************)
			//Calcolo ingombro attuale
			IF NOT TFAsseInFinestra(Posizione_Attuale:=ModuleAx_J^.Ax^.AxRef^.NcToPlc.ActPos,Posizione_Finale:=Mission^.JPick,FinestraDiControllo:=5) THEN //Se la pinza non è già nella finestra di destinazione 
				(* Calcolo l'ingombro massimo che assume durante il ciclo di lavoro nelle direzioni X e Y *)
				(*TFCalcoloIngombroOttimizzatoPinza(  Quota_RotazioneAttuale			:= ModuleAx_J^.Ax^.AxRef^.NcToPlc.ActPos,
													Quota_RotazioneDestinazione		:= Mission^.JPick,
													IngombroSuperficialePinzaMAX	:= IngombroSuperficialePinzaMAX,
													Lunghezza						:= Larghezza,
													Larghezza						:= Lunghezza,
													IngombroOttimizzatoX_InTransito	=> IngombroOttimizzatoX_InTransito,
													IngombroOttimizzatoY_InTransito	=> IngombroOttimizzatoY_InTransito);*)
			ELSE;
				//IngombroOttimizzatoX_InTransito := ABS(IngombroSuperficialePinzaMAX * SIN(deg_to_rad((ATAN(Larghezza/Lunghezza)*1/0.017+ ModuleAx_J^.Ax^.AxRef^.NcToPlc.ActPos)))); //Ingombro Attuale direzione X
				//IngombroOttimizzatoY_InTransito := ABS(IngombroSuperficialePinzaMAX * COS(deg_to_rad((ATAN(Larghezza/Lunghezza)*1/0.017+ ModuleAx_J^.Ax^.AxRef^.NcToPlc.ActPos)))); //Ingombro Attuale direzione Y		
			END_IF
			(* Valutazione colonne in base al verso del pallettizzatore: verso stabilito guardando il pallettizzatore con la linea alle spalle *)
			CASE VERSO_PALLETTIZZATORE OF
				PALLETTIZZATORE_DX :
									TFCalcolaQuotaIngombroColonne(	QuotaY_ColonnaDX						:= WorkFootprint^[6].Y, //DX
																	QuotaY_ColonnaSX						:= WorkFootprint^[5].Y, //SX
																	QuotaAttualeAsse						:= ModuleAX_Y^.Ax^.AxRef^.NcToPlc.ActPos,
																	IngombroOttimizzatoY_InTransito         := IngombroOttimizzatoY_InTransito,
																	OffsetSicurezza_Y						:= OffsetSicurezza_Y,
																	QuotaDestinazioneAsse					:= Mission^.YPick,
																	Pinza_InIngombroColonne_Attuale 		=> Pinza_InIngombroColonne_Attuale,
																	Pinza_InIngombroColonne_Destinazione 	=> Pinza_InIngombroColonne_Destinazione,
																	QuotaFuoriIngombro_Attuale_Y 			=> QuotaFuoriIngombro_Attuale_Y,
																	QuotaFuoriIngombro_Destinazione_Y 		=> QuotaFuoriIngombro_Destinazione_Y);
																	
				PALLETTIZZATORE_SX :
									TFCalcolaQuotaIngombroColonne(	QuotaY_ColonnaDX						:= WorkFootprint^[6].Y, //DX
																	QuotaY_ColonnaSX						:= WorkFootprint^[5].Y, //SX
																	QuotaAttualeAsse						:= ModuleAX_Y^.Ax^.AxRef^.NcToPlc.ActPos,
																	OffsetSicurezza_Y						:= OffsetSicurezza_Y,
																	IngombroOttimizzatoY_InTransito         := IngombroOttimizzatoY_InTransito,
																	QuotaDestinazioneAsse					:= Mission^.YPick,
																	Pinza_InIngombroColonne_Attuale 		=> Pinza_InIngombroColonne_Attuale,
																	Pinza_InIngombroColonne_Destinazione 	=> Pinza_InIngombroColonne_Destinazione,
																	QuotaFuoriIngombro_Attuale_Y 			=> QuotaFuoriIngombro_Attuale_Y,
																	QuotaFuoriIngombro_Destinazione_Y 		=> QuotaFuoriIngombro_Destinazione_Y);
			END_CASE
			
			(* Setto la quota di fuori ingombro che la pinza dovrà assumere durante la traslazione per evitare la collisione con le colonne *)	
			//IF Pinza_InIngombroColonne_Attuale THEN
				QuotaFuoriIngombroColonne_Y := QuotaFuoriIngombro_Attuale_Y;
			//ELSIF Pinza_InIngombroColonne_Destinazione THEN
			//	QuotaFuoriIngombroColonne_Y := QuotaFuoriIngombro_Destinazione_Y;
			//ELSE
			//	QuotaFuoriIngombroColonne_Y := QuotaFuoriIngombro_Attuale_Y;
			//END_IF
			
					
			(* Se sono in ingombro nella posizione attuale o nella posizione di destinazione, devo andare fuori-ingombro con la Y *)
			IF (Pinza_InIngombroColonne_Attuale OR Pinza_InIngombroColonne_Destinazione) THEN 
				IF (AsseXInFinestraDiRiposo AND AsseYInFinestraDiRiposo AND AsseJInFinestraDiRiposo) THEN //Se sono in finestra di riposo con tutti gli assi non devo andare fuori-ingombro con la Y
					FuoriIngombroYNecessarioTMP := FALSE;
				ELSE
					FuoriIngombroYNecessarioTMP := TRUE;
				END_IF
			ELSE
				FuoriIngombroYNecessarioTMP := FALSE;
			END_IF
		END_IF
								
	WAMANAGER_CICLO_RIPOSO_END: 
		CalcolaIngombro := TRUE;
(*			
	WAMANAGER_CICLO_PALL_INIT:
		CalcolaIngombro := TRUE;
	
	WAMANAGER_CICLO_PRELIEVO_PALL_RUN:
		DirezioneXPositiva := TFDirezioneAssePositiva(Posizione_Attuale:=ModuleAX_X^.Ax^.Status.ActPosition,Posizione_Finale:=Mission^.XPick);
		DirezioneXNegativa := NOT DirezioneXPositiva;
		(* Valuto se con l'asse X sono fuori dall'area delle colonne *)
		QuotaX_ConsensoRotazionePinza_Raggiunta := TFPinzaInFuoriIngombroColonne_DirezioneX(DirezioneXPositiva:=DirezioneXPositiva,
																							AsseInMoto:=ModuleAX_X^.Ax^.AxRef^.Status.Moving,
																							PosizioneAttuale:=ModuleAX_X^.Ax^.Status.ActPosition,
																							PosizioneColonna_X:=WorkFootprint^[5].X,  
																							IngombroColonna_X:=WorkFootprint^[5].XDim,
																							IngombroPinza_X:=IngombroX);
				
		IF CalcolaIngombro THEN
			CalcolaIngombro := FALSE;
			(* Definisco il tipo di area in cui si trova a lavorare il pallettizzatore *)
			AreaInLavoroPositiva := FALSE;
			AreaInLavoroNegativa := FALSE;
			AreaInLavoroPositivaNegativa := FALSE; 

			IF (WorkArea^[Mission^.PPick].X >= (WorkFootprint^[5].X + WorkFootprint^[5].XDim)) AND 				//se la piazzola di prelievo è nella campata POSITIVA
				(ModuleAX_X^.Ax^.Status.ActPosition >= (WorkFootprint^[5].X + WorkFootprint^[5].XDim)) THEN // Se la posizione attuale è nella campata POSITIVA
					AreaInLavoroPositiva := TRUE;
			ELSIF (WorkArea^[Mission^.PPick].X <= WorkFootprint^[5].X) AND 			//se la piazzola di prelievo è nella campata NEGATIVA
				(ModuleAX_X^.Ax^.Status.ActPosition <= WorkFootprint^[5].X) THEN 		// Se la posizione attuale è nella campata NEGATIVA
					AreaInLavoroNegativa := TRUE;
			ELSE
				AreaInLavoroPositivaNegativa := TRUE;
			END_IF	
			
			(**************************************************************************************************************************************************)
			(* Ingombro ottimizzato della pinza sul punto di prelievo *)
			(**************************************************************************************************************************************************)
			IngombroOttimizzatoX_InPuntoDiPrelievo := ABS(IngombroSuperficialePinzaMAX * SIN(deg_to_rad((ATAN(Larghezza/Lunghezza)*1/0.017+ Mission^.JPick))));
			IngombroOttimizzatoY_InPuntoDiPrelievo := ABS(IngombroSuperficialePinzaMAX * COS(deg_to_rad((ATAN(Larghezza/Lunghezza)*1/0.017+ Mission^.JPick))));
			(**************************************************************************************************************************************************)
			(* Ingombro ottimizzato della pinza sul punto di deposito *)
			(**************************************************************************************************************************************************)
			IngombroOttimizzatoX_InPuntoDiDeposito := ABS(IngombroSuperficialePinzaMAX * SIN(deg_to_rad((ATAN(Larghezza/Lunghezza)*1/0.017+ Mission^.JPlace))));
			IngombroOttimizzatoY_InPuntoDiDeposito := ABS(IngombroSuperficialePinzaMAX * COS(deg_to_rad((ATAN(Larghezza/Lunghezza)*1/0.017+ Mission^.JPlace))));
						
			(**************************************************************************************************************************************************)
			(**************************************************************************************************************************************************)
			(* Valuto la direzione della X *)
			DirezioneXPositiva := TFDirezioneAssePositiva(Posizione_Attuale:=ModuleAX_X^.Ax^.Status.ActPosition,Posizione_Finale:=Mission^.XPick);
			DirezioneXNegativa := NOT DirezioneXPositiva;
							
			(**************************************************************************************************************************************************)
			(* Ingombro MASSIMO della pinza durante il transito *)
			(**************************************************************************************************************************************************)
			//Calcolo ingombro attuale
			IF NOT TFAsseInFinestra(Posizione_Attuale:=ModuleAx_J^.Ax^.AxRef^.NcToPlc.ActPos,Posizione_Finale:=Mission^.JPick,FinestraDiControllo:=5)  THEN //Se la pinza non è già nella finestra di destinazione 
				(* Calcolo l'ingombro massimo che assume durante il ciclo di lavoro nelle direzioni X e Y *)
				TFCalcoloIngombroOttimizzatoPinza(  Quota_RotazioneAttuale			:= ModuleAx_J^.Ax^.AxRef^.NcToPlc.ActPos,
													Quota_RotazioneDestinazione		:= Mission^.JPick,
													IngombroSuperficialePinzaMAX	:= IngombroSuperficialePinzaMAX,
													Lunghezza						:= Larghezza,
													Larghezza						:= Lunghezza,
													IngombroOttimizzatoX_InTransito	=> IngombroOttimizzatoX_InTransito,
													IngombroOttimizzatoY_InTransito	=> IngombroOttimizzatoY_InTransito);
			ELSE
				IngombroOttimizzatoX_InTransito := ABS(IngombroSuperficialePinzaMAX * SIN(deg_to_rad((ATAN(Larghezza/Lunghezza)*1/0.017+ ModuleAx_J^.Ax^.AxRef^.NcToPlc.ActPos)))); //Ingombro Attuale direzione X
				IngombroOttimizzatoY_InTransito := ABS(IngombroSuperficialePinzaMAX * COS(deg_to_rad((ATAN(Larghezza/Lunghezza)*1/0.017+ ModuleAx_J^.Ax^.AxRef^.NcToPlc.ActPos)))); //Ingombro Attuale direzione Y		
			END_IF
			(* Valutazione colonne in base al verso del pallettizzatore: verso stabilito guardando il pallettizzatore con la linea alle spalle *)
			CASE VERSO_PALLETTIZZATORE OF
				PALLETTIZZATORE_DX :
									TFCalcolaQuotaIngombroColonne(	QuotaY_ColonnaDX						:= WorkFootprint^[6].Y, //DX
																	QuotaY_ColonnaSX						:= WorkFootprint^[5].Y, //SX
																	QuotaAttualeAsse						:= ModuleAX_Y^.Ax^.AxRef^.NcToPlc.ActPos,
																	IngombroOttimizzatoY_InTransito         := IngombroOttimizzatoY_InTransito,
																	OffsetSicurezza_Y						:= OffsetSicurezza_Y,
																	QuotaDestinazioneAsse					:= Mission^.YPick,
																	Pinza_InIngombroColonne_Attuale 		=> Pinza_InIngombroColonne_Attuale,
																	Pinza_InIngombroColonne_Destinazione 	=> Pinza_InIngombroColonne_Destinazione,
																	QuotaFuoriIngombro_Attuale_Y 			=> QuotaFuoriIngombro_Attuale_Y,
																	QuotaFuoriIngombro_Destinazione_Y 		=> QuotaFuoriIngombro_Destinazione_Y);
																	
				PALLETTIZZATORE_SX :
									TFCalcolaQuotaIngombroColonne(	QuotaY_ColonnaDX						:= WorkFootprint^[6].Y, //DX
																	QuotaY_ColonnaSX						:= WorkFootprint^[5].Y, //SX
																	QuotaAttualeAsse						:= ModuleAX_Y^.Ax^.AxRef^.NcToPlc.ActPos,
																	OffsetSicurezza_Y						:= OffsetSicurezza_Y,
																	IngombroOttimizzatoY_InTransito         := IngombroOttimizzatoY_InTransito,
																	QuotaDestinazioneAsse					:= Mission^.YPick,
																	Pinza_InIngombroColonne_Attuale 		=> Pinza_InIngombroColonne_Attuale,
																	Pinza_InIngombroColonne_Destinazione 	=> Pinza_InIngombroColonne_Destinazione,
																	QuotaFuoriIngombro_Attuale_Y 			=> QuotaFuoriIngombro_Attuale_Y,
																	QuotaFuoriIngombro_Destinazione_Y 		=> QuotaFuoriIngombro_Destinazione_Y);
			END_CASE
			
			(* Setto la quota di fuori ingombro che la pinza dovrà assumere durante la traslazione per evitare la collisione con le colonne *)	
			QuotaFuoriIngombroColonne_Y := QuotaFuoriIngombro_Attuale_Y;
					
			(* Se sono in ingombro nella posizione attuale o nella posizione di destinazione, devo andare fuori-ingombro con la Y *)
			IF (Pinza_InIngombroColonne_Attuale OR Pinza_InIngombroColonne_Destinazione) THEN 
				IF (AsseXInFinestraDiRiposo AND AsseYInFinestraDiRiposo AND AsseJInFinestraDiRiposo) THEN //Se sono in finestra di riposo con tutti gli assi non devo andare fuori-ingombro con la Y
					FuoriIngombroYNecessarioTMP := FALSE;
				ELSE
					FuoriIngombroYNecessarioTMP := TRUE;
				END_IF
			ELSE
				FuoriIngombroYNecessarioTMP := FALSE;
			END_IF
		END_IF
		
	WAMANAGER_CICLO_PRELIEVO_PALL_END:
		CalcolaIngombro := TRUE;					
		
	WAMANAGER_CICLO_DEPOSITO_PALL_RUN:
		DirezioneXPositiva := TFDirezioneAssePositiva(Posizione_Attuale:=ModuleAX_X^.Ax^.Status.ActPosition,Posizione_Finale:=Mission^.XPlace);
		DirezioneXNegativa := NOT DirezioneXPositiva;
		(* Valuto se con l'asse X sono fuori dall'area delle colonne *)
		QuotaX_ConsensoRotazionePinza_Raggiunta := TFPinzaInFuoriIngombroColonne_DirezioneX(DirezioneXPositiva:=DirezioneXPositiva,
																							AsseInMoto:=ModuleAX_X^.Ax^.AxRef^.Status.Moving,
																							PosizioneAttuale:=ModuleAX_X^.Ax^.Status.ActPosition,
																							PosizioneColonna_X:=WorkFootprint^[5].X,  
																							IngombroColonna_X:=WorkFootprint^[5].XDim,
																							IngombroPinza_X:=IngombroX);
																					
		IF CalcolaIngombro THEN
			CalcolaIngombro := FALSE;
			(* Definisco il tipo di area in cui si trova a lavorare il pallettizzatore *)
			AreaInLavoroPositiva := FALSE;
			AreaInLavoroNegativa := FALSE;
			AreaInLavoroPositivaNegativa := FALSE; 
			
			IF (WorkArea^[Mission^.PPlace].X >= (WorkFootprint^[5].X + WorkFootprint^[5].XDim)) AND 				//se la piazzola di prelievo è nella campata POSITIVA
				(ModuleAX_X^.Ax^.Status.ActPosition >= (WorkFootprint^[5].X + WorkFootprint^[5].XDim)) THEN // Se la posizione attuale è nella campata POSITIVA
					AreaInLavoroPositiva := TRUE;
			ELSIF (WorkArea^[Mission^.PPlace].X <= WorkFootprint^[5].X) AND 			//se la piazzola di prelievo è nella campata NEGATIVA
				(ModuleAX_X^.Ax^.Status.ActPosition <= WorkFootprint^[5].X) THEN 		// Se la posizione attuale è nella campata NEGATIVA
					AreaInLavoroNegativa := TRUE;
			ELSE
				AreaInLavoroPositivaNegativa := TRUE;
			END_IF
			
			(**************************************************************************************************************************************************)
			(* Ingombro ottimizzato della pinza sul punto di prelievo *)
			(**************************************************************************************************************************************************)
			IngombroOttimizzatoX_InPuntoDiPrelievo := ABS(IngombroSuperficialePinzaMAX * SIN(deg_to_rad((ATAN(Larghezza/Lunghezza)*1/0.017+ Mission^.JPick))));
			IngombroOttimizzatoY_InPuntoDiPrelievo := ABS(IngombroSuperficialePinzaMAX * COS(deg_to_rad((ATAN(Larghezza/Lunghezza)*1/0.017+ Mission^.JPick))));
			(**************************************************************************************************************************************************)
			(* Ingombro ottimizzato della pinza sul punto di deposito *)
			(**************************************************************************************************************************************************)
			IngombroOttimizzatoX_InPuntoDiDeposito := ABS(IngombroSuperficialePinzaMAX * SIN(deg_to_rad((ATAN(Larghezza/Lunghezza)*1/0.017+ Mission^.JPlace))));
			IngombroOttimizzatoY_InPuntoDiDeposito := ABS(IngombroSuperficialePinzaMAX * COS(deg_to_rad((ATAN(Larghezza/Lunghezza)*1/0.017+ Mission^.JPlace))));
						
			(**************************************************************************************************************************************************)
			(**************************************************************************************************************************************************)
			(* Valuto la direzione della X *)
			DirezioneXPositiva := TFDirezioneAssePositiva(Posizione_Attuale:=ModuleAX_X^.Ax^.Status.ActPosition,Posizione_Finale:=Mission^.XPlace);
			DirezioneXNegativa := NOT DirezioneXPositiva;
							
			(**************************************************************************************************************************************************)
			(* Ingombro MASSIMO della pinza durante il transito *)
			(**************************************************************************************************************************************************)
			//Calcolo ingombro attuale
			IF NOT TFAsseInFinestra(Posizione_Attuale:=ModuleAx_J^.Ax^.AxRef^.NcToPlc.ActPos,Posizione_Finale:=Mission^.JPlace,FinestraDiControllo:=5)  THEN //Se la pinza non è già nella finestra di destinazione 
				(* Calcolo l'ingombro massimo che assume durante il ciclo di lavoro nelle direzioni X e Y *)
				TFCalcoloIngombroOttimizzatoPinza(  Quota_RotazioneAttuale			:= ModuleAx_J^.Ax^.AxRef^.NcToPlc.ActPos,
													Quota_RotazioneDestinazione		:= Mission^.JPlace,
													IngombroSuperficialePinzaMAX	:= IngombroSuperficialePinzaMAX,
													Lunghezza						:= Larghezza,
													Larghezza						:= Lunghezza,
													IngombroOttimizzatoX_InTransito	=> IngombroOttimizzatoX_InTransito,
													IngombroOttimizzatoY_InTransito	=> IngombroOttimizzatoY_InTransito);
			ELSE
				IngombroOttimizzatoX_InTransito := ABS(IngombroSuperficialePinzaMAX * SIN(deg_to_rad((ATAN(Larghezza/Lunghezza)*1/0.017+ ModuleAx_J^.Ax^.AxRef^.NcToPlc.ActPos)))); //Ingombro Attuale direzione X
				IngombroOttimizzatoY_InTransito := ABS(IngombroSuperficialePinzaMAX * COS(deg_to_rad((ATAN(Larghezza/Lunghezza)*1/0.017+ ModuleAx_J^.Ax^.AxRef^.NcToPlc.ActPos)))); //Ingombro Attuale direzione Y		
			END_IF
			(* Valutazione colonne in base al verso del pallettizzatore: verso stabilito guardando il pallettizzatore con la linea alle spalle *)
			CASE VERSO_PALLETTIZZATORE OF
				PALLETTIZZATORE_DX :
									TFCalcolaQuotaIngombroColonne(	QuotaY_ColonnaDX						:= WorkFootprint^[6].Y, //DX
																	QuotaY_ColonnaSX						:= WorkFootprint^[5].Y, //SX
																	QuotaAttualeAsse						:= ModuleAX_Y^.Ax^.AxRef^.NcToPlc.ActPos,
																	IngombroOttimizzatoY_InTransito         := IngombroOttimizzatoY_InTransito,
																	OffsetSicurezza_Y						:= OffsetSicurezza_Y,
																	QuotaDestinazioneAsse					:= Mission^.YPlace,
																	Pinza_InIngombroColonne_Attuale 		=> Pinza_InIngombroColonne_Attuale,
																	Pinza_InIngombroColonne_Destinazione 	=> Pinza_InIngombroColonne_Destinazione,
																	QuotaFuoriIngombro_Attuale_Y 			=> QuotaFuoriIngombro_Attuale_Y,
																	QuotaFuoriIngombro_Destinazione_Y 		=> QuotaFuoriIngombro_Destinazione_Y);
																	
				PALLETTIZZATORE_SX :
									TFCalcolaQuotaIngombroColonne(	QuotaY_ColonnaDX						:= WorkFootprint^[6].Y, //DX
																	QuotaY_ColonnaSX						:= WorkFootprint^[5].Y, //SX
																	QuotaAttualeAsse						:= ModuleAX_Y^.Ax^.AxRef^.NcToPlc.ActPos,
																	OffsetSicurezza_Y						:= OffsetSicurezza_Y,
																	IngombroOttimizzatoY_InTransito         := IngombroOttimizzatoY_InTransito,
																	QuotaDestinazioneAsse					:= Mission^.YPlace,
																	Pinza_InIngombroColonne_Attuale 		=> Pinza_InIngombroColonne_Attuale,
																	Pinza_InIngombroColonne_Destinazione 	=> Pinza_InIngombroColonne_Destinazione,
																	QuotaFuoriIngombro_Attuale_Y 			=> QuotaFuoriIngombro_Attuale_Y,
																	QuotaFuoriIngombro_Destinazione_Y 		=> QuotaFuoriIngombro_Destinazione_Y);
			END_CASE
			
			(* Setto la quota di fuori ingombro che la pinza dovrà assumere durante la traslazione per evitare la collisione con le colonne *)	
			QuotaFuoriIngombroColonne_Y := QuotaFuoriIngombro_Attuale_Y;
					
			(* Se sono in ingombro nella posizione attuale o nella posizione di destinazione, devo andare fuori-ingombro con la Y *)
			IF (Pinza_InIngombroColonne_Attuale OR Pinza_InIngombroColonne_Destinazione) THEN 
				IF (AsseXInFinestraDiRiposo AND AsseYInFinestraDiRiposo AND AsseJInFinestraDiRiposo) THEN //Se sono in finestra di riposo con tutti gli assi non devo andare fuori-ingombro con la Y
					FuoriIngombroYNecessarioTMP := FALSE;
				ELSE
					FuoriIngombroYNecessarioTMP := TRUE;
				END_IF
			ELSE
				FuoriIngombroYNecessarioTMP := FALSE;
			END_IF
		END_IF
		
	WAMANAGER_CICLO_DEPOSITO_PALL_END:
		CalcolaIngombro := TRUE;	
	
	WAMANAGER_CICLO_FALDA_VUOTI_INIT:
		CalcolaIngombro := TRUE;	
	
	WAMANAGER_CICLO_PRELIEVO_FALDA_VUOTI_RUN:
		DirezioneXPositiva := TFDirezioneAssePositiva(Posizione_Attuale:=ModuleAX_X^.Ax^.Status.ActPosition,Posizione_Finale:=Mission^.XPick);
		DirezioneXNegativa := NOT DirezioneXPositiva;
		
				
		IF CalcolaIngombro THEN
			CalcolaIngombro := FALSE;
			(* Definisco il tipo di area in cui si trova a lavorare il pallettizzatore *)
			AreaInLavoroPositiva := FALSE;
			AreaInLavoroNegativa := FALSE;
			AreaInLavoroPositivaNegativa := FALSE;

			IF (WorkArea^[Mission^.PPick].X >= (WorkFootprint^[5].X + WorkFootprint^[5].XDim)) AND 				//se la piazzola di prelievo è nella campata POSITIVA
				(ModuleAX_X^.Ax^.Status.ActPosition >= (WorkFootprint^[5].X + WorkFootprint^[5].XDim)) THEN // Se la posizione attuale è nella campata POSITIVA
					AreaInLavoroPositiva := TRUE;
			ELSIF (WorkArea^[Mission^.PPick].X <= WorkFootprint^[5].X) AND 			//se la piazzola di prelievo è nella campata NEGATIVA
				(ModuleAX_X^.Ax^.Status.ActPosition <= WorkFootprint^[5].X) THEN 		// Se la posizione attuale è nella campata NEGATIVA
					AreaInLavoroNegativa := TRUE;
			ELSE
				AreaInLavoroPositivaNegativa := TRUE;
			END_IF 
			
			(**************************************************************************************************************************************************)
			(* Ingombro ottimizzato della pinza sul punto di prelievo *)
			(**************************************************************************************************************************************************)
			IngombroOttimizzatoX_InPuntoDiPrelievo := ABS(IngombroSuperficialePinzaMAX * SIN(deg_to_rad((ATAN(Larghezza/Lunghezza)*1/0.017+ Mission^.JPick))));
			IngombroOttimizzatoY_InPuntoDiPrelievo := ABS(IngombroSuperficialePinzaMAX * COS(deg_to_rad((ATAN(Larghezza/Lunghezza)*1/0.017+ Mission^.JPick))));
			(**************************************************************************************************************************************************)
			(* Ingombro ottimizzato della pinza sul punto di deposito *)
			(**************************************************************************************************************************************************)
			IngombroOttimizzatoX_InPuntoDiDeposito := ABS(IngombroSuperficialePinzaMAX * SIN(deg_to_rad((ATAN(Larghezza/Lunghezza)*1/0.017+ Mission^.JPlace))));
			IngombroOttimizzatoY_InPuntoDiDeposito := ABS(IngombroSuperficialePinzaMAX * COS(deg_to_rad((ATAN(Larghezza/Lunghezza)*1/0.017+ Mission^.JPlace))));
						
			(**************************************************************************************************************************************************)
			(**************************************************************************************************************************************************)
			(* Valuto la direzione della X *)
			DirezioneXPositiva := TFDirezioneAssePositiva(Posizione_Attuale:=ModuleAX_X^.Ax^.Status.ActPosition,Posizione_Finale:=Mission^.XPick);
			DirezioneXNegativa := NOT DirezioneXPositiva;
							
			(**************************************************************************************************************************************************)
			(* Ingombro MASSIMO della pinza durante il transito *)
			(**************************************************************************************************************************************************)
			//Calcolo ingombro attuale
			IF NOT TFAsseInFinestra(Posizione_Attuale:=ModuleAx_J^.Ax^.AxRef^.NcToPlc.ActPos,Posizione_Finale:=Mission^.JPick,FinestraDiControllo:=5)  THEN //Se la pinza non è già nella finestra di destinazione 
				(* Calcolo l'ingombro massimo che assume durante il ciclo di lavoro nelle direzioni X e Y *)
				TFCalcoloIngombroOttimizzatoPinza(  Quota_RotazioneAttuale			:= ModuleAx_J^.Ax^.AxRef^.NcToPlc.ActPos,
													Quota_RotazioneDestinazione		:= Mission^.JPick,
													IngombroSuperficialePinzaMAX	:= IngombroSuperficialePinzaMAX,
													Lunghezza						:= Larghezza,
													Larghezza						:= Lunghezza,
													IngombroOttimizzatoX_InTransito	=> IngombroOttimizzatoX_InTransito,
													IngombroOttimizzatoY_InTransito	=> IngombroOttimizzatoY_InTransito);
			ELSE
				IngombroOttimizzatoX_InTransito := ABS(IngombroSuperficialePinzaMAX * SIN(deg_to_rad((ATAN(Larghezza/Lunghezza)*1/0.017+ ModuleAx_J^.Ax^.AxRef^.NcToPlc.ActPos)))); //Ingombro Attuale direzione X
				IngombroOttimizzatoY_InTransito := ABS(IngombroSuperficialePinzaMAX * COS(deg_to_rad((ATAN(Larghezza/Lunghezza)*1/0.017+ ModuleAx_J^.Ax^.AxRef^.NcToPlc.ActPos)))); //Ingombro Attuale direzione Y		
			END_IF
			(* Valutazione colonne in base al verso del pallettizzatore: verso stabilito guardando il pallettizzatore con la linea alle spalle *)
			CASE VERSO_PALLETTIZZATORE OF
				PALLETTIZZATORE_DX :
									TFCalcolaQuotaIngombroColonne(	QuotaY_ColonnaDX						:= WorkFootprint^[6].Y, //DX
																	QuotaY_ColonnaSX						:= WorkFootprint^[5].Y, //SX
																	QuotaAttualeAsse						:= ModuleAX_Y^.Ax^.AxRef^.NcToPlc.ActPos,
																	IngombroOttimizzatoY_InTransito         := IngombroOttimizzatoY_InTransito,
																	OffsetSicurezza_Y						:= OffsetSicurezza_Y,
																	QuotaDestinazioneAsse					:= Mission^.YPick,
																	Pinza_InIngombroColonne_Attuale 		=> Pinza_InIngombroColonne_Attuale,
																	Pinza_InIngombroColonne_Destinazione 	=> Pinza_InIngombroColonne_Destinazione,
																	QuotaFuoriIngombro_Attuale_Y 			=> QuotaFuoriIngombro_Attuale_Y,
																	QuotaFuoriIngombro_Destinazione_Y 		=> QuotaFuoriIngombro_Destinazione_Y);
																	
				PALLETTIZZATORE_SX :
									TFCalcolaQuotaIngombroColonne(	QuotaY_ColonnaDX						:= WorkFootprint^[6].Y, //DX
																	QuotaY_ColonnaSX						:= WorkFootprint^[5].Y, //SX
																	QuotaAttualeAsse						:= ModuleAX_Y^.Ax^.AxRef^.NcToPlc.ActPos,
																	OffsetSicurezza_Y						:= OffsetSicurezza_Y,
																	IngombroOttimizzatoY_InTransito         := IngombroOttimizzatoY_InTransito,
																	QuotaDestinazioneAsse					:= Mission^.YPick,
																	Pinza_InIngombroColonne_Attuale 		=> Pinza_InIngombroColonne_Attuale,
																	Pinza_InIngombroColonne_Destinazione 	=> Pinza_InIngombroColonne_Destinazione,
																	QuotaFuoriIngombro_Attuale_Y 			=> QuotaFuoriIngombro_Attuale_Y,
																	QuotaFuoriIngombro_Destinazione_Y 		=> QuotaFuoriIngombro_Destinazione_Y);
			END_CASE
			
			(* Setto la quota di fuori ingombro che la pinza dovrà assumere durante la traslazione per evitare la collisione con le colonne *)	
			QuotaFuoriIngombroColonne_Y := QuotaFuoriIngombro_Attuale_Y;
					
			(* Se sono in ingombro nella posizione attuale o nella posizione di destinazione, devo andare fuori-ingombro con la Y *)
			IF (Pinza_InIngombroColonne_Attuale OR Pinza_InIngombroColonne_Destinazione) THEN 
				IF (AsseXInFinestraDiRiposo AND AsseYInFinestraDiRiposo AND AsseJInFinestraDiRiposo) THEN //Se sono in finestra di riposo con tutti gli assi non devo andare fuori-ingombro con la Y
					FuoriIngombroYNecessarioTMP := FALSE;
				ELSE
					FuoriIngombroYNecessarioTMP := TRUE;
				END_IF
			ELSE
				FuoriIngombroYNecessarioTMP := FALSE;
			END_IF
		END_IF
		
		(* Valuto se con l'asse X sono fuori dall'area delle colonne *)
		QuotaX_ConsensoRotazionePinza_Raggiunta := NOT AreaInLavoroPositivaNegativa OR TFPinzaInFuoriIngombroColonne_DirezioneX(DirezioneXPositiva:=DirezioneXPositiva,
																							AsseInMoto:=ModuleAX_X^.Ax^.AxRef^.Status.Moving,
																							PosizioneAttuale:=ModuleAX_X^.Ax^.Status.ActPosition,
																							PosizioneColonna_X:=WorkFootprint^[5].X,  
																							IngombroColonna_X:=WorkFootprint^[5].XDim,
																							IngombroPinza_X:=IngombroX);
			
	WAMANAGER_CICLO_PRELIEVO_FALDA_VUOTI_END:
		CalcolaIngombro := TRUE;	
		
